(* Logix 5000 project; controller VET 1756-L62 rev 19.52; software revision 19.01; part 7 of 27 *)

        [7].Data.flags[2] := 5, [7].Data.flags[3] := 5, [7].Data.flags[4] := 5, [7].Data.flags[5] := 5, [7].Data.flags[6] := 5, [7].Data.flags[7] := 5, [7].Data.flags[8] := 5, [7].Data.fecha_i[0] := 20140324, [7].Data.fecha_i[1] := 20140324, [7].Data.fecha_i[2] := 20140324, [7].Data.fecha_i[3] := 20140324, [7].Data.fecha_i[4] := 20140324, [7].Data.fecha_i[5] := 20140324, [7].Data.fecha_i[6] := 20140324, [7].Data.fecha_i[7] := 20140324, [7].Data.fecha_i[8] := 20140324, [7].Data.fecha_f[0] := 20140324, [7].Data.fecha_f[1] := 20140324, [7].Data.fecha_f[2] := 20140324, [7].Data.fecha_f[3] := 20140324, [7].Data.fecha_f[4] := 20140324, [7].Data.fecha_f[5] := 20140324, [7].Data.fecha_f[6] := 20140324, [7].Data.fecha_f[7] := 20140324, [7].Data.fecha_f[8] := 20140324, [7].Data.hora_i[0] := 11072683, [7].Data.hora_i[1] := 11073663, [7].Data.hora_i[2] := 11072683, [7].Data.hora_i[3] := 11073503, [7].Data.hora_i[4] := 11072683, [7].Data.hora_i[5] := 11074453, [7].Data.hora_i[6] := 11100033, [7].Data.hora_i[7] := 11072683, [7].Data.hora_i[8] := 11073593, [7].Data.hora_f[0] := 11073623, [7].Data.hora_f[1] := 11074913, [7].Data.hora_f[2] := 11073463, [7].Data.hora_f[3] := 11074613, [7].Data.hora_f[4] := 11074413, [7].Data.hora_f[5] := 11075843, [7].Data.hora_f[6] := 11105503, [7].Data.hora_f[7] := 11073553, [7].Data.hora_f[8] := 11074863, [8].Head.folio := 20, [8].Head.orden := -2, [8].Head.formula := 'DUMMY$00$00$00$00$00', [8].Head.estado := 5, [8].Head.correlativo := 10, [8].Head.total_batch := 10, [8].Head.peso_teorico := 1201.0, [8].Data.codigo[0] := 5, [8].Data.codigo[1] := 6, [8].Data.codigo[2] := 7, [8].Data.codigo[3] := 8, [8].Data.codigo[4] := 10, [8].Data.codigo[5] := 20, [8].Data.codigo[6] := 25, [8].Data.codigo[7] := 49, [8].Data.codigo[8] := 50, [8].Data.peso_f[0] := 8.0,
        [8].Data.peso_f[1] := 7.0, [8].Data.peso_f[2] := 6.0, [8].Data.peso_f[3] := 5.0, [8].Data.peso_f[4] := 600.0, [8].Data.peso_f[5] := 400.0, [8].Data.peso_f[6] := 95.0, [8].Data.peso_f[7] := 30.0, [8].Data.peso_f[8] := 50.0, [9].Head.folio := 21, [9].Head.orden := -3, [9].Head.formula := 'DUMMY$00$00$00$00$00', [9].Head.correlativo := 1, [9].Head.total_batch := 20, [9].Head.peso_teorico := 1733.0, [9].Data.codigo[0] := 51, [9].Data.codigo[1] := 53, [9].Data.codigo[2] := 55, [9].Data.codigo[3] := 57, [9].Data.codigo[4] := 60, [9].Data.codigo[5] := 62, [9].Data.codigo[6] := 64, [9].Data.codigo[7] := 66, [9].Data.codigo[8] := 67, [9].Data.codigo[9] := 68, [9].Data.codigo[10] := 69, [9].Data.codigo[11] := 70, [9].Data.codigo[12] := 74, [9].Data.codigo[13] := 75, [9].Data.codigo[14] := 76, [9].Data.codigo[15] := 77, [9].Data.codigo[16] := 81, [9].Data.peso_f[0] := 400.0, [9].Data.peso_f[1] := 350.0, [9].Data.peso_f[2] := 175.0, [9].Data.peso_f[3] := 225.0, [9].Data.peso_f[4] := 125.0, [9].Data.peso_f[5] := 125.0, [9].Data.peso_f[6] := 65.0, [9].Data.peso_f[7] := 65.0, [9].Data.peso_f[8] := 30.0, [9].Data.peso_f[9] := 25.0, [9].Data.peso_f[10] := 17.5, [9].Data.peso_f[11] := 17.5, [9].Data.peso_f[12] := 30.0, [9].Data.peso_f[13] := 5.0, [9].Data.peso_f[14] := 4.0, [9].Data.peso_f[15] := 4.0, [9].Data.peso_f[16] := 70.0, [9].Data.peso_r[0] := 406.2177, [9].Data.peso_r[1] := 352.48218, [9].Data.peso_r[2] := 181.6532, [9].Data.peso_r[3] := 226.84772, [9].Data.peso_r[4] := 129.14812, [9].Data.peso_r[5] := 129.12715, [9].Data.peso_r[6] := 68.647064, [9].Data.peso_r[7] := 68.64438, [9].Data.peso_r[8] := 30.003521, [9].Data.peso_r[9] := 24.965416, [9].Data.peso_r[10] := 17.580997, [9].Data.peso_r[11] := 17.461937,
        [9].Data.peso_r[12] := 30.00344, [9].Data.peso_r[13] := 4.9946327, [9].Data.peso_r[14] := 3.9117737, [9].Data.peso_r[15] := 3.952877, [9].Data.peso_r[16] := 70.002106, [9].Data.tolva[0] := 2, [9].Data.tolva[1] := 4, [9].Data.tolva[2] := 10, [9].Data.tolva[3] := 12, [9].Data.tolva[4] := 7, [9].Data.tolva[5] := 9, [9].Data.tolva[6] := 15, [9].Data.tolva[7] := 17, [9].Data.tolva[8] := 18, [9].Data.tolva[9] := 19, [9].Data.tolva[10] := 20, [9].Data.tolva[11] := 21, [9].Data.tolva[12] := 26, [9].Data.tolva[13] := 27, [9].Data.tolva[14] := 28, [9].Data.tolva[15] := 29, [9].Data.tolva[16] := 38, [9].Data.lugar[0] := 1, [9].Data.lugar[1] := 1, [9].Data.lugar[2] := 1, [9].Data.lugar[3] := 1, [9].Data.lugar[4] := 2, [9].Data.lugar[5] := 2, [9].Data.lugar[6] := 2, [9].Data.lugar[7] := 2, [9].Data.lugar[8] := 3, [9].Data.lugar[9] := 3, [9].Data.lugar[10] := 3, [9].Data.lugar[11] := 3, [9].Data.lugar[12] := 4, [9].Data.lugar[13] := 4, [9].Data.lugar[14] := 4, [9].Data.lugar[15] := 4, [9].Data.lugar[16] := 6, [9].Data.flags[0] := 5, [9].Data.flags[1] := 5, [9].Data.flags[2] := 5, [9].Data.flags[3] := 5, [9].Data.flags[4] := 5, [9].Data.flags[5] := 5, [9].Data.flags[6] := 5, [9].Data.flags[7] := 5, [9].Data.flags[8] := 5, [9].Data.flags[9] := 5, [9].Data.flags[10] := 5, [9].Data.flags[11] := 5, [9].Data.flags[12] := 5, [9].Data.flags[13] := 5, [9].Data.flags[14] := 5, [9].Data.flags[15] := 5, [9].Data.flags[16] := 5, [9].Data.fecha_i[0] := 20140324, [9].Data.fecha_i[1] := 20140324, [9].Data.fecha_i[2] := 20140324, [9].Data.fecha_i[3] := 20140324,
        [9].Data.fecha_i[4] := 20140324, [9].Data.fecha_i[5] := 20140324, [9].Data.fecha_i[6] := 20140324, [9].Data.fecha_i[7] := 20140324, [9].Data.fecha_i[8] := 20140324, [9].Data.fecha_i[9] := 20140324, [9].Data.fecha_i[10] := 20140324, [9].Data.fecha_i[11] := 20140324, [9].Data.fecha_i[12] := 20140324, [9].Data.fecha_i[13] := 20140324, [9].Data.fecha_i[14] := 20140324, [9].Data.fecha_i[15] := 20140324, [9].Data.fecha_i[16] := 20140324, [9].Data.fecha_f[0] := 20140324, [9].Data.fecha_f[1] := 20140324, [9].Data.fecha_f[2] := 20140324, [9].Data.fecha_f[3] := 20140324, [9].Data.fecha_f[4] := 20140324, [9].Data.fecha_f[5] := 20140324, [9].Data.fecha_f[6] := 20140324, [9].Data.fecha_f[7] := 20140324, [9].Data.fecha_f[8] := 20140324, [9].Data.fecha_f[9] := 20140324, [9].Data.fecha_f[10] := 20140324, [9].Data.fecha_f[11] := 20140324, [9].Data.fecha_f[12] := 20140324, [9].Data.fecha_f[13] := 20140324, [9].Data.fecha_f[14] := 20140324, [9].Data.fecha_f[15] := 20140324, [9].Data.fecha_f[16] := 20140324, [9].Data.hora_i[0] := 15282353, [9].Data.hora_i[1] := 15284663, [9].Data.hora_i[2] := 15290343, [9].Data.hora_i[3] := 15292253, [9].Data.hora_i[4] := 15282353, [9].Data.hora_i[5] := 15284903, [9].Data.hora_i[6] := 15290823, [9].Data.hora_i[7] := 15292083, [9].Data.hora_i[8] := 15282353, [9].Data.hora_i[9] := 15311783, [9].Data.hora_i[10] := 15321493, [9].Data.hora_i[11] := 15325653, [9].Data.hora_i[12] := 15282353, [9].Data.hora_i[13] := 15323253, [9].Data.hora_i[14] := 15324993, [9].Data.hora_i[15] := 15330103, [9].Data.hora_i[16] := 15335763, [9].Data.hora_f[0] := 15284623, [9].Data.hora_f[1] := 15290303, [9].Data.hora_f[2] := 15292213, [9].Data.hora_f[3] := 15294183, [9].Data.hora_f[4] := 15284863, [9].Data.hora_f[5] := 15290783, [9].Data.hora_f[6] := 15292043, [9].Data.hora_f[7] := 15293023, [9].Data.hora_f[8] := 15311743, [9].Data.hora_f[9] := 15321453, [9].Data.hora_f[10] := 15325613, [9].Data.hora_f[11] := 15333843, [9].Data.hora_f[12] := 15323213,
        [9].Data.hora_f[13] := 15324953, [9].Data.hora_f[14] := 15330063, [9].Data.hora_f[15] := 15331563, [9].Data.hora_f[16] := 15344023, [10].Head.folio := 22, [10].Head.orden := -3, [10].Head.formula := 'DUMMY$00$00$00$00$00', [10].Head.correlativo := 2, [10].Head.total_batch := 20, [10].Head.peso_teorico := 1733.0, [10].Data.codigo[0] := 51, [10].Data.codigo[1] := 53, [10].Data.codigo[2] := 55, [10].Data.codigo[3] := 57, [10].Data.codigo[4] := 60, [10].Data.codigo[5] := 62, [10].Data.codigo[6] := 64, [10].Data.codigo[7] := 66, [10].Data.codigo[8] := 67, [10].Data.codigo[9] := 68, [10].Data.codigo[10] := 69, [10].Data.codigo[11] := 70, [10].Data.codigo[12] := 74, [10].Data.codigo[13] := 75, [10].Data.codigo[14] := 76, [10].Data.codigo[15] := 77, [10].Data.codigo[16] := 81, [10].Data.peso_f[0] := 400.0, [10].Data.peso_f[1] := 350.0, [10].Data.peso_f[2] := 175.0, [10].Data.peso_f[3] := 225.0, [10].Data.peso_f[4] := 125.0, [10].Data.peso_f[5] := 125.0, [10].Data.peso_f[6] := 65.0, [10].Data.peso_f[7] := 65.0, [10].Data.peso_f[8] := 30.0, [10].Data.peso_f[9] := 25.0, [10].Data.peso_f[10] := 17.5, [10].Data.peso_f[11] := 17.5, [10].Data.peso_f[12] := 30.0, [10].Data.peso_f[13] := 5.0, [10].Data.peso_f[14] := 4.0, [10].Data.peso_f[15] := 4.0, [10].Data.peso_f[16] := 70.0, [10].Data.peso_r[0] := 406.18576, [10].Data.peso_r[1] := 355.42447, [10].Data.peso_r[2] := 181.19794, [10].Data.peso_r[3] := 226.84515, [10].Data.peso_r[4] := 125.444466, [10].Data.peso_r[5] := 127.34431, [10].Data.peso_r[6] := 68.58177, [10].Data.peso_r[7] := 68.6817, [10].Data.peso_r[8] := 30.003046, [10].Data.peso_r[9] := 24.965014, [10].Data.peso_r[10] := 17.42197, [10].Data.peso_r[11] := 17.461983, [10].Data.peso_r[12] := 30.003046, [10].Data.peso_r[13] := 4.995043, [10].Data.peso_r[14] := 3.9528885, [10].Data.peso_r[15] := 3.9532852,
        [10].Data.peso_r[16] := 70.0021, [10].Data.tolva[0] := 2, [10].Data.tolva[1] := 4, [10].Data.tolva[2] := 10, [10].Data.tolva[3] := 12, [10].Data.tolva[4] := 7, [10].Data.tolva[5] := 9, [10].Data.tolva[6] := 15, [10].Data.tolva[7] := 17, [10].Data.tolva[8] := 18, [10].Data.tolva[9] := 19, [10].Data.tolva[10] := 20, [10].Data.tolva[11] := 21, [10].Data.tolva[12] := 26, [10].Data.tolva[13] := 27, [10].Data.tolva[14] := 28, [10].Data.tolva[15] := 29, [10].Data.tolva[16] := 38, [10].Data.lugar[0] := 1, [10].Data.lugar[1] := 1, [10].Data.lugar[2] := 1, [10].Data.lugar[3] := 1, [10].Data.lugar[4] := 2, [10].Data.lugar[5] := 2, [10].Data.lugar[6] := 2, [10].Data.lugar[7] := 2, [10].Data.lugar[8] := 3, [10].Data.lugar[9] := 3, [10].Data.lugar[10] := 3, [10].Data.lugar[11] := 3, [10].Data.lugar[12] := 4, [10].Data.lugar[13] := 4, [10].Data.lugar[14] := 4, [10].Data.lugar[15] := 4, [10].Data.lugar[16] := 6, [10].Data.flags[0] := 5, [10].Data.flags[1] := 5, [10].Data.flags[2] := 5, [10].Data.flags[3] := 5, [10].Data.flags[4] := 5, [10].Data.flags[5] := 5, [10].Data.flags[6] := 5, [10].Data.flags[7] := 5, [10].Data.flags[8] := 5, [10].Data.flags[9] := 5, [10].Data.flags[10] := 5, [10].Data.flags[11] := 5, [10].Data.flags[12] := 5, [10].Data.flags[13] := 5, [10].Data.flags[14] := 5, [10].Data.flags[15] := 5, [10].Data.flags[16] := 5, [10].Data.fecha_i[0] := 20140324, [10].Data.fecha_i[1] := 20140324, [10].Data.fecha_i[2] := 20140324, [10].Data.fecha_i[3] := 20140324, [10].Data.fecha_i[4] := 20140324, [10].Data.fecha_i[5] := 20140324, [10].Data.fecha_i[6] := 20140324, [10].Data.fecha_i[7] := 20140324,
        [10].Data.fecha_i[8] := 20140324, [10].Data.fecha_i[9] := 20140324, [10].Data.fecha_i[10] := 20140324, [10].Data.fecha_i[11] := 20140324, [10].Data.fecha_i[12] := 20140324, [10].Data.fecha_i[13] := 20140324, [10].Data.fecha_i[14] := 20140324, [10].Data.fecha_i[15] := 20140324, [10].Data.fecha_i[16] := 20140324, [10].Data.fecha_f[0] := 20140324, [10].Data.fecha_f[1] := 20140324, [10].Data.fecha_f[2] := 20140324, [10].Data.fecha_f[3] := 20140324, [10].Data.fecha_f[4] := 20140324, [10].Data.fecha_f[5] := 20140324, [10].Data.fecha_f[6] := 20140324, [10].Data.fecha_f[7] := 20140324, [10].Data.fecha_f[8] := 20140324, [10].Data.fecha_f[9] := 20140324, [10].Data.fecha_f[10] := 20140324, [10].Data.fecha_f[11] := 20140324, [10].Data.fecha_f[12] := 20140324, [10].Data.fecha_f[13] := 20140324, [10].Data.fecha_f[14] := 20140324, [10].Data.fecha_f[15] := 20140324, [10].Data.fecha_f[16] := 20140324, [10].Data.hora_i[0] := 15335773, [10].Data.hora_i[1] := 15342253, [10].Data.hora_i[2] := 15402193, [10].Data.hora_i[3] := 15403953, [10].Data.hora_i[4] := 15335773, [10].Data.hora_i[5] := 15340653, [10].Data.hora_i[6] := 15341983, [10].Data.hora_i[7] := 15343023, [10].Data.hora_i[8] := 15335773, [10].Data.hora_i[9] := 15402173, [10].Data.hora_i[10] := 15411913, [10].Data.hora_i[11] := 15415733, [10].Data.hora_i[12] := 15335773, [10].Data.hora_i[13] := 15350103, [10].Data.hora_i[14] := 15402183, [10].Data.hora_i[15] := 15403313, [10].Data.hora_i[16] := 15425823, [10].Data.hora_f[0] := 15342213, [10].Data.hora_f[1] := 15350583, [10].Data.hora_f[2] := 15403913, [10].Data.hora_f[3] := 15405703, [10].Data.hora_f[4] := 15340613, [10].Data.hora_f[5] := 15341943, [10].Data.hora_f[6] := 15342983, [10].Data.hora_f[7] := 15343963, [10].Data.hora_f[8] := 15350063, [10].Data.hora_f[9] := 15411873, [10].Data.hora_f[10] := 15415693, [10].Data.hora_f[11] := 15423913, [10].Data.hora_f[12] := 15350063, [10].Data.hora_f[13] := 15351773, [10].Data.hora_f[14] := 15403273, [10].Data.hora_f[15] := 15404783, [10].Data.hora_f[16] := 15434053,
        [11].Head.folio := 23, [11].Head.orden := -3, [11].Head.formula := 'DUMMY$00$00$00$00$00', [11].Head.correlativo := 3, [11].Head.total_batch := 20, [11].Head.peso_teorico := 1733.0, [11].Data.codigo[0] := 51, [11].Data.codigo[1] := 53, [11].Data.codigo[2] := 55, [11].Data.codigo[3] := 57, [11].Data.codigo[4] := 60, [11].Data.codigo[5] := 62, [11].Data.codigo[6] := 64, [11].Data.codigo[7] := 66, [11].Data.codigo[8] := 67, [11].Data.codigo[9] := 68, [11].Data.codigo[10] := 69, [11].Data.codigo[11] := 70, [11].Data.codigo[12] := 74, [11].Data.codigo[13] := 75, [11].Data.codigo[14] := 76, [11].Data.codigo[15] := 77, [11].Data.codigo[16] := 81, [11].Data.peso_f[0] := 400.0, [11].Data.peso_f[1] := 350.0, [11].Data.peso_f[2] := 175.0, [11].Data.peso_f[3] := 225.0, [11].Data.peso_f[4] := 125.0, [11].Data.peso_f[5] := 125.0, [11].Data.peso_f[6] := 65.0, [11].Data.peso_f[7] := 65.0, [11].Data.peso_f[8] := 30.0, [11].Data.peso_f[9] := 25.0, [11].Data.peso_f[10] := 17.5, [11].Data.peso_f[11] := 17.5, [11].Data.peso_f[12] := 30.0, [11].Data.peso_f[13] := 5.0, [11].Data.peso_f[14] := 4.0, [11].Data.peso_f[15] := 4.0, [11].Data.peso_f[16] := 70.0, [11].Data.peso_r[0] := 400.25983, [11].Data.peso_r[1] := 352.48248, [11].Data.peso_r[2] := 175.69269, [11].Data.peso_r[3] := 226.84637, [11].Data.peso_r[4] := 125.44443, [11].Data.peso_r[5] := 127.34447, [11].Data.peso_r[6] := 66.7538, [11].Data.peso_r[7] := 64.86154, [11].Data.peso_r[8] := 30.003036, [11].Data.peso_r[9] := 25.005493, [11].Data.peso_r[10] := 17.461853, [11].Data.peso_r[11] := 17.462425, [11].Data.peso_r[12] := 30.003036, [11].Data.peso_r[13] := 4.995037, [11].Data.peso_r[14] := 3.9113045, [11].Data.peso_r[15] := 3.9532928, [11].Data.peso_r[16] := 70.0001, [11].Data.tolva[0] := 2, [11].Data.tolva[1] := 4, [11].Data.tolva[2] := 10,
        [11].Data.tolva[3] := 12, [11].Data.tolva[4] := 7, [11].Data.tolva[5] := 9, [11].Data.tolva[6] := 15, [11].Data.tolva[7] := 17, [11].Data.tolva[8] := 18, [11].Data.tolva[9] := 19, [11].Data.tolva[10] := 20, [11].Data.tolva[11] := 21, [11].Data.tolva[12] := 26, [11].Data.tolva[13] := 27, [11].Data.tolva[14] := 28, [11].Data.tolva[15] := 29, [11].Data.tolva[16] := 38, [11].Data.lugar[0] := 1, [11].Data.lugar[1] := 1, [11].Data.lugar[2] := 1, [11].Data.lugar[3] := 1, [11].Data.lugar[4] := 2, [11].Data.lugar[5] := 2, [11].Data.lugar[6] := 2, [11].Data.lugar[7] := 2, [11].Data.lugar[8] := 3, [11].Data.lugar[9] := 3, [11].Data.lugar[10] := 3, [11].Data.lugar[11] := 3, [11].Data.lugar[12] := 4, [11].Data.lugar[13] := 4, [11].Data.lugar[14] := 4, [11].Data.lugar[15] := 4, [11].Data.lugar[16] := 6, [11].Data.flags[0] := 5, [11].Data.flags[1] := 5, [11].Data.flags[2] := 5, [11].Data.flags[3] := 5, [11].Data.flags[4] := 5, [11].Data.flags[5] := 5, [11].Data.flags[6] := 5, [11].Data.flags[7] := 5, [11].Data.flags[8] := 5, [11].Data.flags[9] := 5, [11].Data.flags[10] := 5, [11].Data.flags[11] := 5, [11].Data.flags[12] := 5, [11].Data.flags[13] := 5, [11].Data.flags[14] := 5, [11].Data.flags[15] := 5, [11].Data.flags[16] := 5, [11].Data.fecha_i[0] := 20140324, [11].Data.fecha_i[1] := 20140324, [11].Data.fecha_i[2] := 20140324, [11].Data.fecha_i[3] := 20140324, [11].Data.fecha_i[4] := 20140324, [11].Data.fecha_i[5] := 20140324, [11].Data.fecha_i[6] := 20140324, [11].Data.fecha_i[7] := 20140324, [11].Data.fecha_i[8] := 20140324, [11].Data.fecha_i[9] := 20140324, [11].Data.fecha_i[10] := 20140324, [11].Data.fecha_i[11] := 20140324,
        [11].Data.fecha_i[12] := 20140324, [11].Data.fecha_i[13] := 20140324, [11].Data.fecha_i[14] := 20140324, [11].Data.fecha_i[15] := 20140324, [11].Data.fecha_i[16] := 20140324, [11].Data.fecha_f[0] := 20140324, [11].Data.fecha_f[1] := 20140324, [11].Data.fecha_f[2] := 20140324, [11].Data.fecha_f[3] := 20140324, [11].Data.fecha_f[4] := 20140324, [11].Data.fecha_f[5] := 20140324, [11].Data.fecha_f[6] := 20140324, [11].Data.fecha_f[7] := 20140324, [11].Data.fecha_f[8] := 20140324, [11].Data.fecha_f[9] := 20140324, [11].Data.fecha_f[10] := 20140324, [11].Data.fecha_f[11] := 20140324, [11].Data.fecha_f[12] := 20140324, [11].Data.fecha_f[13] := 20140324, [11].Data.fecha_f[14] := 20140324, [11].Data.fecha_f[15] := 20140324, [11].Data.fecha_f[16] := 20140324, [11].Data.hora_i[0] := 15425833, [11].Data.hora_i[1] := 15431183, [11].Data.hora_i[2] := 15454413, [11].Data.hora_i[3] := 15455193, [11].Data.hora_i[4] := 15425833, [11].Data.hora_i[5] := 15430713, [11].Data.hora_i[6] := 15454423, [11].Data.hora_i[7] := 15455843, [11].Data.hora_i[8] := 15425833, [11].Data.hora_i[9] := 15440173, [11].Data.hora_i[10] := 15445913, [11].Data.hora_i[11] := 15453733, [11].Data.hora_i[12] := 15425833, [11].Data.hora_i[13] := 15440163, [11].Data.hora_i[14] := 15441903, [11].Data.hora_i[15] := 15443023, [11].Data.hora_i[16] := 15481743, [11].Data.hora_f[0] := 15431143, [11].Data.hora_f[1] := 15454373, [11].Data.hora_f[2] := 15455153, [11].Data.hora_f[3] := 15472663, [11].Data.hora_f[4] := 15430673, [11].Data.hora_f[5] := 15454383, [11].Data.hora_f[6] := 15455803, [11].Data.hora_f[7] := 15460433, [11].Data.hora_f[8] := 15440123, [11].Data.hora_f[9] := 15445873, [11].Data.hora_f[10] := 15453693, [11].Data.hora_f[11] := 15461933, [11].Data.hora_f[12] := 15440123, [11].Data.hora_f[13] := 15441863, [11].Data.hora_f[14] := 15442983, [11].Data.hora_f[15] := 15444513, [11].Data.hora_f[16] := 15485973, [12].Head.folio := 24, [12].Head.orden := -3, [12].Head.formula := 'DUMMY$00$00$00$00$00', [12].Head.correlativo := 4,
        [12].Head.total_batch := 20, [12].Head.peso_teorico := 1733.0, [12].Data.codigo[0] := 51, [12].Data.codigo[1] := 53, [12].Data.codigo[2] := 55, [12].Data.codigo[3] := 57, [12].Data.codigo[4] := 60, [12].Data.codigo[5] := 62, [12].Data.codigo[6] := 64, [12].Data.codigo[7] := 66, [12].Data.codigo[8] := 67, [12].Data.codigo[9] := 68, [12].Data.codigo[10] := 69, [12].Data.codigo[11] := 70, [12].Data.codigo[12] := 74, [12].Data.codigo[13] := 75, [12].Data.codigo[14] := 76, [12].Data.codigo[15] := 77, [12].Data.codigo[16] := 81, [12].Data.peso_f[0] := 400.0, [12].Data.peso_f[1] := 350.0, [12].Data.peso_f[2] := 175.0, [12].Data.peso_f[3] := 225.0, [12].Data.peso_f[4] := 125.0, [12].Data.peso_f[5] := 125.0, [12].Data.peso_f[6] := 65.0, [12].Data.peso_f[7] := 65.0, [12].Data.peso_f[8] := 30.0, [12].Data.peso_f[9] := 25.0, [12].Data.peso_f[10] := 17.5, [12].Data.peso_f[11] := 17.5, [12].Data.peso_f[12] := 30.0, [12].Data.peso_f[13] := 5.0, [12].Data.peso_f[14] := 4.0, [12].Data.peso_f[15] := 4.0, [12].Data.peso_f[16] := 70.0, [12].Data.peso_r[0] := 400.2613, [12].Data.peso_r[1] := 352.48242, [12].Data.peso_r[2] := 175.88062, [12].Data.peso_r[3] := 229.9057, [12].Data.peso_r[4] := 125.44438, [12].Data.peso_r[5] := 127.34422, [12].Data.peso_r[6] := 64.84152, [12].Data.peso_r[7] := 64.861115, [12].Data.peso_r[8] := 30.003, [12].Data.peso_r[9] := 25.005491, [12].Data.peso_r[10] := 17.461853, [12].Data.peso_r[11] := 17.461967, [12].Data.peso_r[12] := 30.003, [12].Data.peso_r[13] := 4.9950314, [12].Data.peso_r[14] := 3.9931755, [12].Data.peso_r[15] := 3.9945488, [12].Data.peso_r[16] := 70.000114, [12].Data.tolva[0] := 2, [12].Data.tolva[1] := 4, [12].Data.tolva[2] := 10, [12].Data.tolva[3] := 12, [12].Data.tolva[4] := 7, [12].Data.tolva[5] := 9, [12].Data.tolva[6] := 15,
        [12].Data.tolva[7] := 17, [12].Data.tolva[8] := 18, [12].Data.tolva[9] := 19, [12].Data.tolva[10] := 20, [12].Data.tolva[11] := 21, [12].Data.tolva[12] := 26, [12].Data.tolva[13] := 27, [12].Data.tolva[14] := 28, [12].Data.tolva[15] := 29, [12].Data.tolva[16] := 38, [12].Data.lugar[0] := 1, [12].Data.lugar[1] := 1, [12].Data.lugar[2] := 1, [12].Data.lugar[3] := 1, [12].Data.lugar[4] := 2, [12].Data.lugar[5] := 2, [12].Data.lugar[6] := 2, [12].Data.lugar[7] := 2, [12].Data.lugar[8] := 3, [12].Data.lugar[9] := 3, [12].Data.lugar[10] := 3, [12].Data.lugar[11] := 3, [12].Data.lugar[12] := 4, [12].Data.lugar[13] := 4, [12].Data.lugar[14] := 4, [12].Data.lugar[15] := 4, [12].Data.lugar[16] := 6, [12].Data.flags[0] := 5, [12].Data.flags[1] := 5, [12].Data.flags[2] := 5, [12].Data.flags[3] := 5, [12].Data.flags[4] := 5, [12].Data.flags[5] := 5, [12].Data.flags[6] := 5, [12].Data.flags[7] := 5, [12].Data.flags[8] := 5, [12].Data.flags[9] := 5, [12].Data.flags[10] := 5, [12].Data.flags[11] := 5, [12].Data.flags[12] := 5, [12].Data.flags[13] := 5, [12].Data.flags[14] := 5, [12].Data.flags[15] := 5, [12].Data.flags[16] := 5, [12].Data.fecha_i[0] := 20140324, [12].Data.fecha_i[1] := 20140324, [12].Data.fecha_i[2] := 20140324, [12].Data.fecha_i[3] := 20140324, [12].Data.fecha_i[4] := 20140324, [12].Data.fecha_i[5] := 20140324, [12].Data.fecha_i[6] := 20140324, [12].Data.fecha_i[7] := 20140324, [12].Data.fecha_i[8] := 20140324, [12].Data.fecha_i[9] := 20140324, [12].Data.fecha_i[10] := 20140324, [12].Data.fecha_i[11] := 20140324, [12].Data.fecha_i[12] := 20140324, [12].Data.fecha_i[13] := 20140324, [12].Data.fecha_i[14] := 20140324, [12].Data.fecha_i[15] := 20140324,
        [12].Data.fecha_i[16] := 20140324, [12].Data.fecha_f[0] := 20140324, [12].Data.fecha_f[1] := 20140324, [12].Data.fecha_f[2] := 20140324, [12].Data.fecha_f[3] := 20140324, [12].Data.fecha_f[4] := 20140324, [12].Data.fecha_f[5] := 20140324, [12].Data.fecha_f[6] := 20140324, [12].Data.fecha_f[7] := 20140324, [12].Data.fecha_f[8] := 20140324, [12].Data.fecha_f[9] := 20140324, [12].Data.fecha_f[10] := 20140324, [12].Data.fecha_f[11] := 20140324, [12].Data.fecha_f[12] := 20140324, [12].Data.fecha_f[13] := 20140324, [12].Data.fecha_f[14] := 20140324, [12].Data.fecha_f[15] := 20140324, [12].Data.fecha_f[16] := 20140324, [12].Data.hora_i[0] := 15481753, [12].Data.hora_i[1] := 15483103, [12].Data.hora_i[2] := 15484333, [12].Data.hora_i[3] := 15485113, [12].Data.hora_i[4] := 15481753, [12].Data.hora_i[5] := 15482633, [12].Data.hora_i[6] := 15510173, [12].Data.hora_i[7] := 15510803, [12].Data.hora_i[8] := 15481753, [12].Data.hora_i[9] := 15492093, [12].Data.hora_i[10] := 15501833, [12].Data.hora_i[11] := 15505663, [12].Data.hora_i[12] := 15481753, [12].Data.hora_i[13] := 15492083, [12].Data.hora_i[14] := 15493823, [12].Data.hora_i[15] := 15494953, [12].Data.hora_i[16] := 15515733, [12].Data.hora_f[0] := 15483063, [12].Data.hora_f[1] := 15484293, [12].Data.hora_f[2] := 15485073, [12].Data.hora_f[3] := 15485993, [12].Data.hora_f[4] := 15482593, [12].Data.hora_f[5] := 15510133, [12].Data.hora_f[6] := 15510763, [12].Data.hora_f[7] := 15511393, [12].Data.hora_f[8] := 15492043, [12].Data.hora_f[9] := 15501793, [12].Data.hora_f[10] := 15505623, [12].Data.hora_f[11] := 15513853, [12].Data.hora_f[12] := 15492043, [12].Data.hora_f[13] := 15493783, [12].Data.hora_f[14] := 15494913, [12].Data.hora_f[15] := 15500473, [12].Data.hora_f[16] := 15523963, [13].Head.folio := 25, [13].Head.orden := -3, [13].Head.formula := 'DUMMY$00$00$00$00$00', [13].Head.correlativo := 5, [13].Head.total_batch := 20, [13].Head.peso_teorico := 1733.0, [13].Data.codigo[0] := 51, [13].Data.codigo[1] := 53,
        [13].Data.codigo[2] := 55, [13].Data.codigo[3] := 57, [13].Data.codigo[4] := 60, [13].Data.codigo[5] := 62, [13].Data.codigo[6] := 64, [13].Data.codigo[7] := 66, [13].Data.codigo[8] := 67, [13].Data.codigo[9] := 68, [13].Data.codigo[10] := 69, [13].Data.codigo[11] := 70, [13].Data.codigo[12] := 74, [13].Data.codigo[13] := 75, [13].Data.codigo[14] := 76, [13].Data.codigo[15] := 77, [13].Data.codigo[16] := 81, [13].Data.peso_f[0] := 400.0, [13].Data.peso_f[1] := 350.0, [13].Data.peso_f[2] := 175.0, [13].Data.peso_f[3] := 225.0, [13].Data.peso_f[4] := 125.0, [13].Data.peso_f[5] := 125.0, [13].Data.peso_f[6] := 65.0, [13].Data.peso_f[7] := 65.0, [13].Data.peso_f[8] := 30.0, [13].Data.peso_f[9] := 25.0, [13].Data.peso_f[10] := 17.5, [13].Data.peso_f[11] := 17.5, [13].Data.peso_f[12] := 30.0, [13].Data.peso_f[13] := 5.0, [13].Data.peso_f[14] := 4.0, [13].Data.peso_f[15] := 4.0, [13].Data.peso_f[16] := 70.0, [13].Data.peso_r[0] := 400.2615, [13].Data.peso_r[1] := 352.48227, [13].Data.peso_r[2] := 175.8805, [13].Data.peso_r[3] := 226.84717, [13].Data.peso_r[4] := 125.44438, [13].Data.peso_r[5] := 127.34419, [13].Data.peso_r[6] := 66.67056, [13].Data.peso_r[7] := 64.86157, [13].Data.peso_r[8] := 30.003036, [13].Data.peso_r[9] := 24.987019, [13].Data.peso_r[10] := 17.463833, [13].Data.peso_r[11] := 17.492538, [13].Data.peso_r[12] := 30.003036, [13].Data.peso_r[13] := 4.9950447, [13].Data.peso_r[14] := 3.9935875, [13].Data.peso_r[15] := 3.9949074, [13].Data.peso_r[16] := 69.50179, [13].Data.tolva[0] := 2, [13].Data.tolva[1] := 4, [13].Data.tolva[2] := 10, [13].Data.tolva[3] := 12, [13].Data.tolva[4] := 7, [13].Data.tolva[5] := 9, [13].Data.tolva[6] := 15, [13].Data.tolva[7] := 17, [13].Data.tolva[8] := 18, [13].Data.tolva[9] := 19, [13].Data.tolva[10] := 20,
        [13].Data.tolva[11] := 21, [13].Data.tolva[12] := 26, [13].Data.tolva[13] := 27, [13].Data.tolva[14] := 28, [13].Data.tolva[15] := 29, [13].Data.tolva[16] := 38, [13].Data.lugar[0] := 1, [13].Data.lugar[1] := 1, [13].Data.lugar[2] := 1, [13].Data.lugar[3] := 1, [13].Data.lugar[4] := 2, [13].Data.lugar[5] := 2, [13].Data.lugar[6] := 2, [13].Data.lugar[7] := 2, [13].Data.lugar[8] := 3, [13].Data.lugar[9] := 3, [13].Data.lugar[10] := 3, [13].Data.lugar[11] := 3, [13].Data.lugar[12] := 4, [13].Data.lugar[13] := 4, [13].Data.lugar[14] := 4, [13].Data.lugar[15] := 4, [13].Data.lugar[16] := 6, [13].Data.flags[0] := 5, [13].Data.flags[1] := 5, [13].Data.flags[2] := 5, [13].Data.flags[3] := 5, [13].Data.flags[4] := 5, [13].Data.flags[5] := 5, [13].Data.flags[6] := 5, [13].Data.flags[7] := 5, [13].Data.flags[8] := 5, [13].Data.flags[9] := 5, [13].Data.flags[10] := 5, [13].Data.flags[11] := 5, [13].Data.flags[12] := 5, [13].Data.flags[13] := 5, [13].Data.flags[14] := 5, [13].Data.flags[15] := 5, [13].Data.flags[16] := 5, [13].Data.fecha_i[0] := 20140324, [13].Data.fecha_i[1] := 20140324, [13].Data.fecha_i[2] := 20140324, [13].Data.fecha_i[3] := 20140324, [13].Data.fecha_i[4] := 20140324, [13].Data.fecha_i[5] := 20140324, [13].Data.fecha_i[6] := 20140324, [13].Data.fecha_i[7] := 20140324, [13].Data.fecha_i[8] := 20140324, [13].Data.fecha_i[9] := 20140324, [13].Data.fecha_i[10] := 20140324, [13].Data.fecha_i[11] := 20140324, [13].Data.fecha_i[12] := 20140324, [13].Data.fecha_i[13] := 20140324, [13].Data.fecha_i[14] := 20140324, [13].Data.fecha_i[15] := 20140324, [13].Data.fecha_i[16] := 20140324, [13].Data.fecha_f[0] := 20140324, [13].Data.fecha_f[1] := 20140324, [13].Data.fecha_f[2] := 20140324,
        [13].Data.fecha_f[3] := 20140324, [13].Data.fecha_f[4] := 20140324, [13].Data.fecha_f[5] := 20140324, [13].Data.fecha_f[6] := 20140324, [13].Data.fecha_f[7] := 20140324, [13].Data.fecha_f[8] := 20140324, [13].Data.fecha_f[9] := 20140324, [13].Data.fecha_f[10] := 20140324, [13].Data.fecha_f[11] := 20140324, [13].Data.fecha_f[12] := 20140324, [13].Data.fecha_f[13] := 20140324, [13].Data.fecha_f[14] := 20140324, [13].Data.fecha_f[15] := 20140324, [13].Data.fecha_f[16] := 20140324, [13].Data.hora_i[0] := 15515743, [13].Data.hora_i[1] := 15521093, [13].Data.hora_i[2] := 15522323, [13].Data.hora_i[3] := 15523113, [13].Data.hora_i[4] := 15515743, [13].Data.hora_i[5] := 15520623, [13].Data.hora_i[6] := 15523103, [13].Data.hora_i[7] := 15524343, [13].Data.hora_i[8] := 15515743, [13].Data.hora_i[9] := 15530083, [13].Data.hora_i[10] := 15535769, [13].Data.hora_i[11] := 15543579, [13].Data.hora_i[12] := 15515743, [13].Data.hora_i[13] := 15530073, [13].Data.hora_i[14] := 15531783, [13].Data.hora_i[15] := 15532913, [13].Data.hora_i[16] := 15553579, [13].Data.hora_f[0] := 15521053, [13].Data.hora_f[1] := 15522283, [13].Data.hora_f[2] := 15523063, [13].Data.hora_f[3] := 15523993, [13].Data.hora_f[4] := 15520583, [13].Data.hora_f[5] := 15523063, [13].Data.hora_f[6] := 15524303, [13].Data.hora_f[7] := 15524933, [13].Data.hora_f[8] := 15530033, [13].Data.hora_f[9] := 15535749, [13].Data.hora_f[10] := 15543559, [13].Data.hora_f[11] := 15551764, [13].Data.hora_f[12] := 15530033, [13].Data.hora_f[13] := 15531743, [13].Data.hora_f[14] := 15532873, [13].Data.hora_f[15] := 15534433, [13].Data.hora_f[16] := 15561754, [14].Head.folio := 26, [14].Head.orden := -3, [14].Head.formula := 'DUMMY$00$00$00$00$00', [14].Head.correlativo := 6, [14].Head.total_batch := 20, [14].Head.peso_teorico := 1733.0, [14].Data.codigo[0] := 51, [14].Data.codigo[1] := 53, [14].Data.codigo[2] := 55, [14].Data.codigo[3] := 57, [14].Data.codigo[4] := 60, [14].Data.codigo[5] := 62,
        [14].Data.codigo[6] := 64, [14].Data.codigo[7] := 66, [14].Data.codigo[8] := 67, [14].Data.codigo[9] := 68, [14].Data.codigo[10] := 69, [14].Data.codigo[11] := 70, [14].Data.codigo[12] := 74, [14].Data.codigo[13] := 75, [14].Data.codigo[14] := 76, [14].Data.codigo[15] := 77, [14].Data.codigo[16] := 81, [14].Data.peso_f[0] := 400.0, [14].Data.peso_f[1] := 350.0, [14].Data.peso_f[2] := 175.0, [14].Data.peso_f[3] := 225.0, [14].Data.peso_f[4] := 125.0, [14].Data.peso_f[5] := 125.0, [14].Data.peso_f[6] := 65.0, [14].Data.peso_f[7] := 65.0, [14].Data.peso_f[8] := 30.0, [14].Data.peso_f[9] := 25.0, [14].Data.peso_f[10] := 17.5, [14].Data.peso_f[11] := 17.5, [14].Data.peso_f[12] := 30.0, [14].Data.peso_f[13] := 5.0, [14].Data.peso_f[14] := 4.0, [14].Data.peso_f[15] := 4.0, [14].Data.peso_f[16] := 70.0, [14].Data.peso_r[0] := 405.18765, [14].Data.peso_r[1] := 347.0085, [14].Data.peso_r[2] := 172.9342, [14].Data.peso_r[3] := 221.31152, [14].Data.peso_r[4] := 125.07125, [14].Data.peso_r[5] := 127.7055, [14].Data.peso_r[6] := 67.87331, [14].Data.peso_r[7] := 65.28912, [14].Data.peso_r[8] := 29.954077, [14].Data.peso_r[9] := 24.973166, [14].Data.peso_r[10] := 17.489925, [14].Data.peso_r[11] := 17.490517, [14].Data.peso_r[12] := 29.954084, [14].Data.peso_r[13] := 4.965147, [14].Data.peso_r[14] := 3.9367218, [14].Data.peso_r[15] := 3.9845467, [14].Data.peso_r[16] := 69.8018, [14].Data.tolva[0] := 2, [14].Data.tolva[1] := 4, [14].Data.tolva[2] := 10, [14].Data.tolva[3] := 12, [14].Data.tolva[4] := 7, [14].Data.tolva[5] := 9, [14].Data.tolva[6] := 15, [14].Data.tolva[7] := 17, [14].Data.tolva[8] := 18, [14].Data.tolva[9] := 19, [14].Data.tolva[10] := 20, [14].Data.tolva[11] := 21, [14].Data.tolva[12] := 26, [14].Data.tolva[13] := 27, [14].Data.tolva[14] := 28,
        [14].Data.tolva[15] := 29, [14].Data.tolva[16] := 38, [14].Data.lugar[0] := 1, [14].Data.lugar[1] := 1, [14].Data.lugar[2] := 1, [14].Data.lugar[3] := 1, [14].Data.lugar[4] := 2, [14].Data.lugar[5] := 2, [14].Data.lugar[6] := 2, [14].Data.lugar[7] := 2, [14].Data.lugar[8] := 3, [14].Data.lugar[9] := 3, [14].Data.lugar[10] := 3, [14].Data.lugar[11] := 3, [14].Data.lugar[12] := 4, [14].Data.lugar[13] := 4, [14].Data.lugar[14] := 4, [14].Data.lugar[15] := 4, [14].Data.lugar[16] := 6, [14].Data.flags[0] := 5, [14].Data.flags[1] := 5, [14].Data.flags[2] := 5, [14].Data.flags[3] := 5, [14].Data.flags[4] := 5, [14].Data.flags[5] := 5, [14].Data.flags[6] := 5, [14].Data.flags[7] := 5, [14].Data.flags[8] := 5, [14].Data.flags[9] := 5, [14].Data.flags[10] := 5, [14].Data.flags[11] := 5, [14].Data.flags[12] := 5, [14].Data.flags[13] := 5, [14].Data.flags[14] := 5, [14].Data.flags[15] := 5, [14].Data.flags[16] := 5, [14].Data.fecha_i[0] := 20140324, [14].Data.fecha_i[1] := 20140324, [14].Data.fecha_i[2] := 20140324, [14].Data.fecha_i[3] := 20140324, [14].Data.fecha_i[4] := 20140324, [14].Data.fecha_i[5] := 20140324, [14].Data.fecha_i[6] := 20140324, [14].Data.fecha_i[7] := 20140324, [14].Data.fecha_i[8] := 20140324, [14].Data.fecha_i[9] := 20140324, [14].Data.fecha_i[10] := 20140324, [14].Data.fecha_i[11] := 20140324, [14].Data.fecha_i[12] := 20140324, [14].Data.fecha_i[13] := 20140324, [14].Data.fecha_i[14] := 20140324, [14].Data.fecha_i[15] := 20140324, [14].Data.fecha_i[16] := 20140324, [14].Data.fecha_f[0] := 20140324, [14].Data.fecha_f[1] := 20140324, [14].Data.fecha_f[2] := 20140324, [14].Data.fecha_f[3] := 20140324, [14].Data.fecha_f[4] := 20140324, [14].Data.fecha_f[5] := 20140324, [14].Data.fecha_f[6] := 20140324,
        [14].Data.fecha_f[7] := 20140324, [14].Data.fecha_f[8] := 20140324, [14].Data.fecha_f[9] := 20140324, [14].Data.fecha_f[10] := 20140324, [14].Data.fecha_f[11] := 20140324, [14].Data.fecha_f[12] := 20140324, [14].Data.fecha_f[13] := 20140324, [14].Data.fecha_f[14] := 20140324, [14].Data.fecha_f[15] := 20140324, [14].Data.fecha_f[16] := 20140324, [14].Data.hora_i[0] := 15553584, [14].Data.hora_i[1] := 15560269, [14].Data.hora_i[2] := 15561464, [14].Data.hora_i[3] := 15562219, [14].Data.hora_i[4] := 15553584, [14].Data.hora_i[5] := 15554444, [14].Data.hora_i[6] := 15561879, [14].Data.hora_i[7] := 15563379, [14].Data.hora_i[8] := 15553584, [14].Data.hora_i[9] := 15563899, [14].Data.hora_i[10] := 15573609, [14].Data.hora_i[11] := 15581424, [14].Data.hora_i[12] := 15553584, [14].Data.hora_i[13] := 15563894, [14].Data.hora_i[14] := 15565604, [14].Data.hora_i[15] := 15570709, [14].Data.hora_i[16] := 15591434, [14].Data.hora_f[0] := 15560249, [14].Data.hora_f[1] := 15561444, [14].Data.hora_f[2] := 15562199, [14].Data.hora_f[3] := 15563089, [14].Data.hora_f[4] := 15554424, [14].Data.hora_f[5] := 15561859, [14].Data.hora_f[6] := 15563359, [14].Data.hora_f[7] := 15563959, [14].Data.hora_f[8] := 15563879, [14].Data.hora_f[9] := 15573589, [14].Data.hora_f[10] := 15581404, [14].Data.hora_f[11] := 15585604, [14].Data.hora_f[12] := 15563874, [14].Data.hora_f[13] := 15565584, [14].Data.hora_f[14] := 15570689, [14].Data.hora_f[15] := 15572179, [14].Data.hora_f[16] := 15595649, [15].Head.folio := 27, [15].Head.orden := -3, [15].Head.formula := 'DUMMY$00$00$00$00$00', [15].Head.correlativo := 7, [15].Head.total_batch := 20, [15].Head.peso_teorico := 1733.0, [15].Data.codigo[0] := 51, [15].Data.codigo[1] := 53, [15].Data.codigo[2] := 55, [15].Data.codigo[3] := 57, [15].Data.codigo[4] := 60, [15].Data.codigo[5] := 62, [15].Data.codigo[6] := 64, [15].Data.codigo[7] := 66, [15].Data.codigo[8] := 67, [15].Data.codigo[9] := 68,
        [15].Data.codigo[10] := 69, [15].Data.codigo[11] := 70, [15].Data.codigo[12] := 74, [15].Data.codigo[13] := 75, [15].Data.codigo[14] := 76, [15].Data.codigo[15] := 77, [15].Data.codigo[16] := 81, [15].Data.peso_f[0] := 400.0, [15].Data.peso_f[1] := 350.0, [15].Data.peso_f[2] := 175.0, [15].Data.peso_f[3] := 225.0, [15].Data.peso_f[4] := 125.0, [15].Data.peso_f[5] := 125.0, [15].Data.peso_f[6] := 65.0, [15].Data.peso_f[7] := 65.0, [15].Data.peso_f[8] := 30.0, [15].Data.peso_f[9] := 25.0, [15].Data.peso_f[10] := 17.5, [15].Data.peso_f[11] := 17.5, [15].Data.peso_f[12] := 30.0, [15].Data.peso_f[13] := 5.0, [15].Data.peso_f[14] := 4.0, [15].Data.peso_f[15] := 4.0, [15].Data.peso_f[16] := 70.0, [15].Data.peso_r[0] := 397.91046, [15].Data.peso_r[1] := 348.57037, [15].Data.peso_r[2] := 173.35175, [15].Data.peso_r[3] := 224.36798, [15].Data.peso_r[4] := 125.071434, [15].Data.peso_r[5] := 128.56516, [15].Data.peso_r[6] := 65.05693, [15].Data.peso_r[7] := 65.05704, [15].Data.peso_r[8] := 29.974127, [15].Data.peso_r[9] := 24.973959, [15].Data.peso_r[10] := 17.489887, [15].Data.peso_r[11] := 17.489935, [15].Data.peso_r[12] := 29.967981, [15].Data.peso_r[13] := 4.9850006, [15].Data.peso_r[14] := 4.004406, [15].Data.peso_r[15] := 4.004547, [15].Data.peso_r[16] := 69.80179, [15].Data.tolva[0] := 2, [15].Data.tolva[1] := 4, [15].Data.tolva[2] := 10, [15].Data.tolva[3] := 12, [15].Data.tolva[4] := 7, [15].Data.tolva[5] := 9, [15].Data.tolva[6] := 15, [15].Data.tolva[7] := 17, [15].Data.tolva[8] := 18, [15].Data.tolva[9] := 19, [15].Data.tolva[10] := 20, [15].Data.tolva[11] := 29, [15].Data.tolva[12] := 26, [15].Data.tolva[13] := 27, [15].Data.tolva[14] := 28, [15].Data.tolva[15] := 21, [15].Data.tolva[16] := 38, [15].Data.lugar[0] := 1, [15].Data.lugar[1] := 1,
        [15].Data.lugar[2] := 1, [15].Data.lugar[3] := 1, [15].Data.lugar[4] := 2, [15].Data.lugar[5] := 2, [15].Data.lugar[6] := 2, [15].Data.lugar[7] := 2, [15].Data.lugar[8] := 3, [15].Data.lugar[9] := 3, [15].Data.lugar[10] := 3, [15].Data.lugar[11] := 4, [15].Data.lugar[12] := 4, [15].Data.lugar[13] := 4, [15].Data.lugar[14] := 4, [15].Data.lugar[15] := 3, [15].Data.lugar[16] := 6, [15].Data.flags[0] := 5, [15].Data.flags[1] := 5, [15].Data.flags[2] := 5, [15].Data.flags[3] := 5, [15].Data.flags[4] := 5, [15].Data.flags[5] := 5, [15].Data.flags[6] := 5, [15].Data.flags[7] := 5, [15].Data.flags[8] := 5, [15].Data.flags[9] := 5, [15].Data.flags[10] := 5, [15].Data.flags[11] := 5, [15].Data.flags[12] := 5, [15].Data.flags[13] := 5, [15].Data.flags[14] := 5, [15].Data.flags[15] := 5, [15].Data.flags[16] := 5, [15].Data.fecha_i[0] := 20140324, [15].Data.fecha_i[1] := 20140324, [15].Data.fecha_i[2] := 20140324, [15].Data.fecha_i[3] := 20140324, [15].Data.fecha_i[4] := 20140324, [15].Data.fecha_i[5] := 20140324, [15].Data.fecha_i[6] := 20140324, [15].Data.fecha_i[7] := 20140324, [15].Data.fecha_i[8] := 20140324, [15].Data.fecha_i[9] := 20140324, [15].Data.fecha_i[10] := 20140324, [15].Data.fecha_i[11] := 20140324, [15].Data.fecha_i[12] := 20140324, [15].Data.fecha_i[13] := 20140324, [15].Data.fecha_i[14] := 20140324, [15].Data.fecha_i[15] := 20140324, [15].Data.fecha_i[16] := 20140324, [15].Data.fecha_f[0] := 20140324, [15].Data.fecha_f[1] := 20140324, [15].Data.fecha_f[2] := 20140324, [15].Data.fecha_f[3] := 20140324, [15].Data.fecha_f[4] := 20140324, [15].Data.fecha_f[5] := 20140324, [15].Data.fecha_f[6] := 20140324, [15].Data.fecha_f[7] := 20140324, [15].Data.fecha_f[8] := 20140324, [15].Data.fecha_f[9] := 20140324, [15].Data.fecha_f[10] := 20140324,
        [15].Data.fecha_f[11] := 20140324, [15].Data.fecha_f[12] := 20140324, [15].Data.fecha_f[13] := 20140324, [15].Data.fecha_f[14] := 20140324, [15].Data.fecha_f[15] := 20140324, [15].Data.fecha_f[16] := 20140324, [15].Data.hora_i[0] := 15592024, [15].Data.hora_i[1] := 15593359, [15].Data.hora_i[2] := 15594569, [15].Data.hora_i[3] := 15595324, [15].Data.hora_i[4] := 15592024, [15].Data.hora_i[5] := 15592884, [15].Data.hora_i[6] := 15595739, [15].Data.hora_i[7] := 16000339, [15].Data.hora_i[8] := 15592024, [15].Data.hora_i[9] := 16002344, [15].Data.hora_i[10] := 16012049, [15].Data.hora_i[11] := 15592024, [15].Data.hora_i[12] := 16000219, [15].Data.hora_i[13] := 16010524, [15].Data.hora_i[14] := 16012204, [15].Data.hora_i[15] := 16015864, [15].Data.hora_i[16] := 16023129, [15].Data.hora_f[0] := 15593339, [15].Data.hora_f[1] := 15594549, [15].Data.hora_f[2] := 15595304, [15].Data.hora_f[3] := 16000199, [15].Data.hora_f[4] := 15592864, [15].Data.hora_f[5] := 15595719, [15].Data.hora_f[6] := 16000319, [15].Data.hora_f[7] := 16000914, [15].Data.hora_f[8] := 16002324, [15].Data.hora_f[9] := 16012029, [15].Data.hora_f[10] := 16015844, [15].Data.hora_f[11] := 16000199, [15].Data.hora_f[12] := 16010504, [15].Data.hora_f[13] := 16012184, [15].Data.hora_f[14] := 16013309, [15].Data.hora_f[15] := 16021349, [15].Data.hora_f[16] := 16031334, [16].Head.folio := 28, [16].Head.orden := -3, [16].Head.formula := 'DUMMY$00$00$00$00$00', [16].Head.correlativo := 8, [16].Head.total_batch := 20, [16].Head.peso_teorico := 1733.0, [16].Data.codigo[0] := 51, [16].Data.codigo[1] := 53, [16].Data.codigo[2] := 55, [16].Data.codigo[3] := 57, [16].Data.codigo[4] := 60, [16].Data.codigo[5] := 62, [16].Data.codigo[6] := 64, [16].Data.codigo[7] := 66, [16].Data.codigo[8] := 67, [16].Data.codigo[9] := 68, [16].Data.codigo[10] := 69, [16].Data.codigo[11] := 70, [16].Data.codigo[12] := 74, [16].Data.codigo[13] := 75,
        [16].Data.codigo[14] := 76, [16].Data.codigo[15] := 77, [16].Data.codigo[16] := 81, [16].Data.peso_f[0] := 400.0, [16].Data.peso_f[1] := 350.0, [16].Data.peso_f[2] := 175.0, [16].Data.peso_f[3] := 225.0, [16].Data.peso_f[4] := 125.0, [16].Data.peso_f[5] := 125.0, [16].Data.peso_f[6] := 65.0, [16].Data.peso_f[7] := 65.0, [16].Data.peso_f[8] := 30.0, [16].Data.peso_f[9] := 25.0, [16].Data.peso_f[10] := 17.5, [16].Data.peso_f[11] := 17.5, [16].Data.peso_f[12] := 30.0, [16].Data.peso_f[13] := 5.0, [16].Data.peso_f[14] := 4.0, [16].Data.peso_f[15] := 4.0, [16].Data.peso_f[16] := 70.0, [16].Data.peso_r[0] := 399.41638, [16].Data.peso_r[1] := 349.9532, [16].Data.peso_r[2] := 173.44592, [16].Data.peso_r[3] := 224.35333, [16].Data.peso_r[4] := 125.06888, [16].Data.peso_r[5] := 127.59076, [16].Data.peso_r[6] := 67.95871, [16].Data.peso_r[7] := 65.37213, [16].Data.peso_r[8] := 29.973724, [16].Data.peso_r[9] := 25.01252, [16].Data.peso_r[10] := 17.487335, [16].Data.peso_r[11] := 17.487408, [16].Data.peso_r[12] := 29.970356, [16].Data.peso_r[13] := 4.9825974, [16].Data.peso_r[14] := 4.00441, [16].Data.peso_r[15] := 4.0045547, [16].Data.peso_r[16] := 70.10178, [16].Data.tolva[0] := 2, [16].Data.tolva[1] := 4, [16].Data.tolva[2] := 10, [16].Data.tolva[3] := 12, [16].Data.tolva[4] := 7, [16].Data.tolva[5] := 9, [16].Data.tolva[6] := 15, [16].Data.tolva[7] := 17, [16].Data.tolva[8] := 18, [16].Data.tolva[9] := 19, [16].Data.tolva[10] := 20, [16].Data.tolva[11] := 29, [16].Data.tolva[12] := 26, [16].Data.tolva[13] := 27, [16].Data.tolva[14] := 28, [16].Data.tolva[15] := 21, [16].Data.tolva[16] := 38, [16].Data.lugar[0] := 1, [16].Data.lugar[1] := 1, [16].Data.lugar[2] := 1, [16].Data.lugar[3] := 1, [16].Data.lugar[4] := 2, [16].Data.lugar[5] := 2,
        [16].Data.lugar[6] := 2, [16].Data.lugar[7] := 2, [16].Data.lugar[8] := 3, [16].Data.lugar[9] := 3, [16].Data.lugar[10] := 3, [16].Data.lugar[11] := 4, [16].Data.lugar[12] := 4, [16].Data.lugar[13] := 4, [16].Data.lugar[14] := 4, [16].Data.lugar[15] := 3, [16].Data.lugar[16] := 6, [16].Data.flags[0] := 5, [16].Data.flags[1] := 5, [16].Data.flags[2] := 5, [16].Data.flags[3] := 5, [16].Data.flags[4] := 5, [16].Data.flags[5] := 5, [16].Data.flags[6] := 5, [16].Data.flags[7] := 5, [16].Data.flags[8] := 5, [16].Data.flags[9] := 5, [16].Data.flags[10] := 5, [16].Data.flags[11] := 5, [16].Data.flags[12] := 5, [16].Data.flags[13] := 5, [16].Data.flags[14] := 5, [16].Data.flags[15] := 5, [16].Data.flags[16] := 5, [16].Data.fecha_i[0] := 20140324, [16].Data.fecha_i[1] := 20140324, [16].Data.fecha_i[2] := 20140324, [16].Data.fecha_i[3] := 20140324, [16].Data.fecha_i[4] := 20140324, [16].Data.fecha_i[5] := 20140324, [16].Data.fecha_i[6] := 20140324, [16].Data.fecha_i[7] := 20140324, [16].Data.fecha_i[8] := 20140324, [16].Data.fecha_i[9] := 20140324, [16].Data.fecha_i[10] := 20140324, [16].Data.fecha_i[11] := 20140324, [16].Data.fecha_i[12] := 20140324, [16].Data.fecha_i[13] := 20140324, [16].Data.fecha_i[14] := 20140324, [16].Data.fecha_i[15] := 20140324, [16].Data.fecha_i[16] := 20140324, [16].Data.fecha_f[0] := 20140324, [16].Data.fecha_f[1] := 20140324, [16].Data.fecha_f[2] := 20140324, [16].Data.fecha_f[3] := 20140324, [16].Data.fecha_f[4] := 20140324, [16].Data.fecha_f[5] := 20140324, [16].Data.fecha_f[6] := 20140324, [16].Data.fecha_f[7] := 20140324, [16].Data.fecha_f[8] := 20140324, [16].Data.fecha_f[9] := 20140324, [16].Data.fecha_f[10] := 20140324, [16].Data.fecha_f[11] := 20140324, [16].Data.fecha_f[12] := 20140324, [16].Data.fecha_f[13] := 20140324, [16].Data.fecha_f[14] := 20140324,
        [16].Data.fecha_f[15] := 20140324, [16].Data.fecha_f[16] := 20140324, [16].Data.hora_i[0] := 16023134, [16].Data.hora_i[1] := 16024474, [16].Data.hora_i[2] := 16025684, [16].Data.hora_i[3] := 16030449, [16].Data.hora_i[4] := 16023134, [16].Data.hora_i[5] := 16023994, [16].Data.hora_i[6] := 16030364, [16].Data.hora_i[7] := 16032219, [16].Data.hora_i[8] := 16023134, [16].Data.hora_i[9] := 16033449, [16].Data.hora_i[10] := 16043169, [16].Data.hora_i[11] := 16023134, [16].Data.hora_i[12] := 16031344, [16].Data.hora_i[13] := 16041654, [16].Data.hora_i[14] := 16043359, [16].Data.hora_i[15] := 16050984, [16].Data.hora_i[16] := 16054269, [16].Data.hora_f[0] := 16024454, [16].Data.hora_f[1] := 16025664, [16].Data.hora_f[2] := 16030429, [16].Data.hora_f[3] := 16031314, [16].Data.hora_f[4] := 16023974, [16].Data.hora_f[5] := 16030344, [16].Data.hora_f[6] := 16032199, [16].Data.hora_f[7] := 16032804, [16].Data.hora_f[8] := 16033429, [16].Data.hora_f[9] := 16043149, [16].Data.hora_f[10] := 16050964, [16].Data.hora_f[11] := 16031324, [16].Data.hora_f[12] := 16041634, [16].Data.hora_f[13] := 16043339, [16].Data.hora_f[14] := 16044464, [16].Data.hora_f[15] := 16052469, [16].Data.hora_f[16] := 16062494, [17].Head.folio := 29, [17].Head.orden := -3, [17].Head.formula := 'DUMMY$00$00$00$00$00', [17].Head.correlativo := 9, [17].Head.total_batch := 20, [17].Head.peso_teorico := 1733.0, [17].Data.codigo[0] := 51, [17].Data.codigo[1] := 53, [17].Data.codigo[2] := 55, [17].Data.codigo[3] := 57, [17].Data.codigo[4] := 60, [17].Data.codigo[5] := 62, [17].Data.codigo[6] := 64, [17].Data.codigo[7] := 66, [17].Data.codigo[8] := 67, [17].Data.codigo[9] := 68, [17].Data.codigo[10] := 69, [17].Data.codigo[11] := 70, [17].Data.codigo[12] := 74, [17].Data.codigo[13] := 75, [17].Data.codigo[14] := 76, [17].Data.codigo[15] := 77, [17].Data.codigo[16] := 81, [17].Data.peso_f[0] := 400.0,
        [17].Data.peso_f[1] := 350.0, [17].Data.peso_f[2] := 175.0, [17].Data.peso_f[3] := 225.0, [17].Data.peso_f[4] := 125.0, [17].Data.peso_f[5] := 125.0, [17].Data.peso_f[6] := 65.0, [17].Data.peso_f[7] := 65.0, [17].Data.peso_f[8] := 30.0, [17].Data.peso_f[9] := 25.0, [17].Data.peso_f[10] := 17.5, [17].Data.peso_f[11] := 17.5, [17].Data.peso_f[12] := 30.0, [17].Data.peso_f[13] := 5.0, [17].Data.peso_f[14] := 4.0, [17].Data.peso_f[15] := 4.0, [17].Data.peso_f[16] := 70.0, [17].Data.peso_r[0] := 399.41718, [17].Data.peso_r[1] := 349.64966, [17].Data.peso_r[2] := 175.0708, [17].Data.peso_r[3] := 225.98505, [17].Data.peso_r[4] := 125.06839, [17].Data.peso_r[5] := 127.61029, [17].Data.peso_r[6] := 65.37216, [17].Data.peso_r[7] := 65.37247, [17].Data.peso_r[8] := 29.994556, [17].Data.peso_r[9] := 25.012424, [17].Data.peso_r[10] := 17.509384, [17].Data.peso_r[11] := 17.509583, [17].Data.peso_r[12] := 29.994267, [17].Data.peso_r[13] := 4.9850388, [17].Data.peso_r[14] := 3.9845657, [17].Data.peso_r[15] := 4.0021057, [17].Data.peso_r[16] := 70.09979, [17].Data.tolva[0] := 2, [17].Data.tolva[1] := 4, [17].Data.tolva[2] := 10, [17].Data.tolva[3] := 12, [17].Data.tolva[4] := 7, [17].Data.tolva[5] := 9, [17].Data.tolva[6] := 15, [17].Data.tolva[7] := 17, [17].Data.tolva[8] := 18, [17].Data.tolva[9] := 19, [17].Data.tolva[10] := 20, [17].Data.tolva[11] := 29, [17].Data.tolva[12] := 26, [17].Data.tolva[13] := 27, [17].Data.tolva[14] := 28, [17].Data.tolva[15] := 21, [17].Data.tolva[16] := 38, [17].Data.lugar[0] := 1, [17].Data.lugar[1] := 1, [17].Data.lugar[2] := 1, [17].Data.lugar[3] := 1, [17].Data.lugar[4] := 2, [17].Data.lugar[5] := 2, [17].Data.lugar[6] := 2, [17].Data.lugar[7] := 2, [17].Data.lugar[8] := 3, [17].Data.lugar[9] := 3,
        [17].Data.lugar[10] := 3, [17].Data.lugar[11] := 4, [17].Data.lugar[12] := 4, [17].Data.lugar[13] := 4, [17].Data.lugar[14] := 4, [17].Data.lugar[15] := 3, [17].Data.lugar[16] := 6, [17].Data.flags[0] := 5, [17].Data.flags[1] := 5, [17].Data.flags[2] := 5, [17].Data.flags[3] := 5, [17].Data.flags[4] := 5, [17].Data.flags[5] := 5, [17].Data.flags[6] := 5, [17].Data.flags[7] := 5, [17].Data.flags[8] := 5, [17].Data.flags[9] := 5, [17].Data.flags[10] := 5, [17].Data.flags[11] := 5, [17].Data.flags[12] := 5, [17].Data.flags[13] := 5, [17].Data.flags[14] := 5, [17].Data.flags[15] := 5, [17].Data.flags[16] := 5, [17].Data.fecha_i[0] := 20140324, [17].Data.fecha_i[1] := 20140324, [17].Data.fecha_i[2] := 20140324, [17].Data.fecha_i[3] := 20140324, [17].Data.fecha_i[4] := 20140324, [17].Data.fecha_i[5] := 20140324, [17].Data.fecha_i[6] := 20140324, [17].Data.fecha_i[7] := 20140324, [17].Data.fecha_i[8] := 20140324, [17].Data.fecha_i[9] := 20140324, [17].Data.fecha_i[10] := 20140324, [17].Data.fecha_i[11] := 20140324, [17].Data.fecha_i[12] := 20140324, [17].Data.fecha_i[13] := 20140324, [17].Data.fecha_i[14] := 20140324, [17].Data.fecha_i[15] := 20140324, [17].Data.fecha_i[16] := 20140324, [17].Data.fecha_f[0] := 20140324, [17].Data.fecha_f[1] := 20140324, [17].Data.fecha_f[2] := 20140324, [17].Data.fecha_f[3] := 20140324, [17].Data.fecha_f[4] := 20140324, [17].Data.fecha_f[5] := 20140324, [17].Data.fecha_f[6] := 20140324, [17].Data.fecha_f[7] := 20140324, [17].Data.fecha_f[8] := 20140324, [17].Data.fecha_f[9] := 20140324, [17].Data.fecha_f[10] := 20140324, [17].Data.fecha_f[11] := 20140324, [17].Data.fecha_f[12] := 20140324, [17].Data.fecha_f[13] := 20140324, [17].Data.fecha_f[14] := 20140324, [17].Data.fecha_f[15] := 20140324, [17].Data.fecha_f[16] := 20140324, [17].Data.hora_i[0] := 16054274, [17].Data.hora_i[1] := 16055619,
        [17].Data.hora_i[2] := 16060824, [17].Data.hora_i[3] := 16061594, [17].Data.hora_i[4] := 16054274, [17].Data.hora_i[5] := 16055134, [17].Data.hora_i[6] := 16061499, [17].Data.hora_i[7] := 16062104, [17].Data.hora_i[8] := 16054274, [17].Data.hora_i[9] := 16064594, [17].Data.hora_i[10] := 16074289, [17].Data.hora_i[11] := 16054274, [17].Data.hora_i[12] := 16062474, [17].Data.hora_i[13] := 16072794, [17].Data.hora_i[14] := 16074489, [17].Data.hora_i[15] := 16082109, [17].Data.hora_i[16] := 16085394, [17].Data.hora_f[0] := 16055599, [17].Data.hora_f[1] := 16060804, [17].Data.hora_f[2] := 16061574, [17].Data.hora_f[3] := 16062469, [17].Data.hora_f[4] := 16055114, [17].Data.hora_f[5] := 16061479, [17].Data.hora_f[6] := 16062084, [17].Data.hora_f[7] := 16062689, [17].Data.hora_f[8] := 16064574, [17].Data.hora_f[9] := 16074269, [17].Data.hora_f[10] := 16082089, [17].Data.hora_f[11] := 16062454, [17].Data.hora_f[12] := 16072774, [17].Data.hora_f[13] := 16074469, [17].Data.hora_f[14] := 16075584, [17].Data.hora_f[15] := 16083599, [17].Data.hora_f[16] := 16093619, [18].Head.folio := 30, [18].Head.orden := -3, [18].Head.formula := 'DUMMY$00$00$00$00$00', [18].Head.correlativo := 10, [18].Head.total_batch := 20, [18].Head.peso_teorico := 1733.0, [18].Data.codigo[0] := 51, [18].Data.codigo[1] := 53, [18].Data.codigo[2] := 55, [18].Data.codigo[3] := 57, [18].Data.codigo[4] := 60, [18].Data.codigo[5] := 62, [18].Data.codigo[6] := 64, [18].Data.codigo[7] := 66, [18].Data.codigo[8] := 67, [18].Data.codigo[9] := 68, [18].Data.codigo[10] := 69, [18].Data.codigo[11] := 70, [18].Data.codigo[12] := 74, [18].Data.codigo[13] := 75, [18].Data.codigo[14] := 76, [18].Data.codigo[15] := 77, [18].Data.codigo[16] := 81, [18].Data.peso_f[0] := 400.0, [18].Data.peso_f[1] := 350.0, [18].Data.peso_f[2] := 175.0, [18].Data.peso_f[3] := 225.0, [18].Data.peso_f[4] := 125.0,
        [18].Data.peso_f[5] := 125.0, [18].Data.peso_f[6] := 65.0, [18].Data.peso_f[7] := 65.0, [18].Data.peso_f[8] := 30.0, [18].Data.peso_f[9] := 25.0, [18].Data.peso_f[10] := 17.5, [18].Data.peso_f[11] := 17.5, [18].Data.peso_f[12] := 30.0, [18].Data.peso_f[13] := 5.0, [18].Data.peso_f[14] := 4.0, [18].Data.peso_f[15] := 4.0, [18].Data.peso_f[16] := 70.0, [18].Data.peso_r[0] := 399.51053, [18].Data.peso_r[1] := 350.04776, [18].Data.peso_r[2] := 175.08862, [18].Data.peso_r[3] := 224.45184, [18].Data.peso_r[4] := 125.070755, [18].Data.peso_r[5] := 125.97429, [18].Data.peso_r[6] := 67.07645, [18].Data.peso_r[7] := 65.28821, [18].Data.peso_r[8] := 29.994556, [18].Data.peso_r[9] := 25.01247, [18].Data.peso_r[10] := 17.506996, [18].Data.peso_r[11] := 17.489944, [18].Data.peso_r[12] := 30.008419, [18].Data.peso_r[13] := 5.005974, [18].Data.peso_r[14] := 4.0019455, [18].Data.peso_r[15] := 4.0045395, [18].Data.peso_r[16] := 69.80178, [18].Data.tolva[0] := 2, [18].Data.tolva[1] := 4, [18].Data.tolva[2] := 10, [18].Data.tolva[3] := 12, [18].Data.tolva[4] := 7, [18].Data.tolva[5] := 9, [18].Data.tolva[6] := 15, [18].Data.tolva[7] := 17, [18].Data.tolva[8] := 18, [18].Data.tolva[9] := 19, [18].Data.tolva[10] := 20, [18].Data.tolva[11] := 29, [18].Data.tolva[12] := 26, [18].Data.tolva[13] := 27, [18].Data.tolva[14] := 28, [18].Data.tolva[15] := 21, [18].Data.tolva[16] := 38, [18].Data.lugar[0] := 1, [18].Data.lugar[1] := 1, [18].Data.lugar[2] := 1, [18].Data.lugar[3] := 1, [18].Data.lugar[4] := 2, [18].Data.lugar[5] := 2, [18].Data.lugar[6] := 2, [18].Data.lugar[7] := 2, [18].Data.lugar[8] := 3, [18].Data.lugar[9] := 3, [18].Data.lugar[10] := 3, [18].Data.lugar[11] := 4, [18].Data.lugar[12] := 4, [18].Data.lugar[13] := 4,
        [18].Data.lugar[14] := 4, [18].Data.lugar[15] := 3, [18].Data.lugar[16] := 6, [18].Data.flags[0] := 5, [18].Data.flags[1] := 5, [18].Data.flags[2] := 5, [18].Data.flags[3] := 5, [18].Data.flags[4] := 5, [18].Data.flags[5] := 5, [18].Data.flags[6] := 5, [18].Data.flags[7] := 5, [18].Data.flags[8] := 5, [18].Data.flags[9] := 5, [18].Data.flags[10] := 5, [18].Data.flags[11] := 5, [18].Data.flags[12] := 5, [18].Data.flags[13] := 5, [18].Data.flags[14] := 5, [18].Data.flags[15] := 5, [18].Data.flags[16] := 5, [18].Data.fecha_i[0] := 20140324, [18].Data.fecha_i[1] := 20140324, [18].Data.fecha_i[2] := 20140324, [18].Data.fecha_i[3] := 20140324, [18].Data.fecha_i[4] := 20140324, [18].Data.fecha_i[5] := 20140324, [18].Data.fecha_i[6] := 20140324, [18].Data.fecha_i[7] := 20140324, [18].Data.fecha_i[8] := 20140324, [18].Data.fecha_i[9] := 20140324, [18].Data.fecha_i[10] := 20140324, [18].Data.fecha_i[11] := 20140324, [18].Data.fecha_i[12] := 20140324, [18].Data.fecha_i[13] := 20140324, [18].Data.fecha_i[14] := 20140324, [18].Data.fecha_i[15] := 20140324, [18].Data.fecha_i[16] := 20140324, [18].Data.fecha_f[0] := 20140324, [18].Data.fecha_f[1] := 20140324, [18].Data.fecha_f[2] := 20140324, [18].Data.fecha_f[3] := 20140324, [18].Data.fecha_f[4] := 20140324, [18].Data.fecha_f[5] := 20140324, [18].Data.fecha_f[6] := 20140324, [18].Data.fecha_f[7] := 20140324, [18].Data.fecha_f[8] := 20140324, [18].Data.fecha_f[9] := 20140324, [18].Data.fecha_f[10] := 20140324, [18].Data.fecha_f[11] := 20140324, [18].Data.fecha_f[12] := 20140324, [18].Data.fecha_f[13] := 20140324, [18].Data.fecha_f[14] := 20140324, [18].Data.fecha_f[15] := 20140324, [18].Data.fecha_f[16] := 20140324, [18].Data.hora_i[0] := 16085399, [18].Data.hora_i[1] := 16090739, [18].Data.hora_i[2] := 16091949, [18].Data.hora_i[3] := 16092709, [18].Data.hora_i[4] := 16085399, [18].Data.hora_i[5] := 16090259,
        [18].Data.hora_i[6] := 16092869, [18].Data.hora_i[7] := 16094579, [18].Data.hora_i[8] := 16085399, [18].Data.hora_i[9] := 16095724, [18].Data.hora_i[10] := 16105449, [18].Data.hora_i[11] := 16085399, [18].Data.hora_i[12] := 16093579, [18].Data.hora_i[13] := 16103894, [18].Data.hora_i[14] := 16105614, [18].Data.hora_i[15] := 16113269, [18].Data.hora_i[16] := 16120549, [18].Data.hora_f[0] := 16090719, [18].Data.hora_f[1] := 16091929, [18].Data.hora_f[2] := 16092689, [18].Data.hora_f[3] := 16093574, [18].Data.hora_f[4] := 16090239, [18].Data.hora_f[5] := 16092849, [18].Data.hora_f[6] := 16094559, [18].Data.hora_f[7] := 16095159, [18].Data.hora_f[8] := 16095704, [18].Data.hora_f[9] := 16105429, [18].Data.hora_f[10] := 16113249, [18].Data.hora_f[11] := 16093559, [18].Data.hora_f[12] := 16103874, [18].Data.hora_f[13] := 16105594, [18].Data.hora_f[14] := 16110714, [18].Data.hora_f[15] := 16114749, [18].Data.hora_f[16] := 16124774, [19].Head.folio := 31, [19].Head.orden := -3, [19].Head.formula := 'DUMMY$00$00$00$00$00', [19].Head.correlativo := 11, [19].Head.total_batch := 20, [19].Head.peso_teorico := 1733.0, [19].Data.codigo[0] := 51, [19].Data.codigo[1] := 53, [19].Data.codigo[2] := 55, [19].Data.codigo[3] := 57, [19].Data.codigo[4] := 60, [19].Data.codigo[5] := 62, [19].Data.codigo[6] := 64, [19].Data.codigo[7] := 66, [19].Data.codigo[8] := 67, [19].Data.codigo[9] := 68, [19].Data.codigo[10] := 69, [19].Data.codigo[11] := 70, [19].Data.codigo[12] := 74, [19].Data.codigo[13] := 75, [19].Data.codigo[14] := 76, [19].Data.codigo[15] := 77, [19].Data.codigo[16] := 81, [19].Data.peso_f[0] := 400.0, [19].Data.peso_f[1] := 350.0, [19].Data.peso_f[2] := 175.0, [19].Data.peso_f[3] := 225.0, [19].Data.peso_f[4] := 125.0, [19].Data.peso_f[5] := 125.0, [19].Data.peso_f[6] := 65.0, [19].Data.peso_f[7] := 65.0, [19].Data.peso_f[8] := 30.0,
        [19].Data.peso_f[9] := 25.0, [19].Data.peso_f[10] := 17.5, [19].Data.peso_f[11] := 17.5, [19].Data.peso_f[12] := 30.0, [19].Data.peso_f[13] := 5.0, [19].Data.peso_f[14] := 4.0, [19].Data.peso_f[15] := 4.0, [19].Data.peso_f[16] := 70.0, [19].Data.peso_r[0] := 398.48602, [19].Data.peso_r[1] := 348.9485, [19].Data.peso_r[2] := 173.54315, [19].Data.peso_r[3] := 223.7793, [19].Data.peso_r[4] := 124.72148, [19].Data.peso_r[5] := 124.674255, [19].Data.peso_r[6] := 67.09276, [19].Data.peso_r[7] := 67.11923, [19].Data.peso_r[8] := 29.992178, [19].Data.peso_r[9] := 25.012426, [19].Data.peso_r[10] := 17.488514, [19].Data.peso_r[11] := 17.50958, [19].Data.peso_r[12] := 29.992468, [19].Data.peso_r[13] := 4.9850464, [19].Data.peso_r[14] := 4.0044594, [19].Data.peso_r[15] := 4.0021286, [19].Data.peso_r[16] := 70.101776, [19].Data.tolva[0] := 2, [19].Data.tolva[1] := 4, [19].Data.tolva[2] := 10, [19].Data.tolva[3] := 12, [19].Data.tolva[4] := 7, [19].Data.tolva[5] := 9, [19].Data.tolva[6] := 15, [19].Data.tolva[7] := 17, [19].Data.tolva[8] := 18, [19].Data.tolva[9] := 19, [19].Data.tolva[10] := 20, [19].Data.tolva[11] := 29, [19].Data.tolva[12] := 26, [19].Data.tolva[13] := 27, [19].Data.tolva[14] := 28, [19].Data.tolva[15] := 21, [19].Data.tolva[16] := 38, [19].Data.lugar[0] := 1, [19].Data.lugar[1] := 1, [19].Data.lugar[2] := 1, [19].Data.lugar[3] := 1, [19].Data.lugar[4] := 2, [19].Data.lugar[5] := 2, [19].Data.lugar[6] := 2, [19].Data.lugar[7] := 2, [19].Data.lugar[8] := 3, [19].Data.lugar[9] := 3, [19].Data.lugar[10] := 3, [19].Data.lugar[11] := 4, [19].Data.lugar[12] := 4, [19].Data.lugar[13] := 4, [19].Data.lugar[14] := 4, [19].Data.lugar[15] := 3, [19].Data.lugar[16] := 6, [19].Data.flags[0] := 5,
        [19].Data.flags[1] := 5, [19].Data.flags[2] := 5, [19].Data.flags[3] := 5, [19].Data.flags[4] := 5, [19].Data.flags[5] := 5, [19].Data.flags[6] := 5, [19].Data.flags[7] := 5, [19].Data.flags[8] := 5, [19].Data.flags[9] := 5, [19].Data.flags[10] := 5, [19].Data.flags[11] := 5, [19].Data.flags[12] := 5, [19].Data.flags[13] := 5, [19].Data.flags[14] := 5, [19].Data.flags[15] := 5, [19].Data.flags[16] := 5, [19].Data.fecha_i[0] := 20140324, [19].Data.fecha_i[1] := 20140324, [19].Data.fecha_i[2] := 20140324, [19].Data.fecha_i[3] := 20140324, [19].Data.fecha_i[4] := 20140324, [19].Data.fecha_i[5] := 20140324, [19].Data.fecha_i[6] := 20140324, [19].Data.fecha_i[7] := 20140324, [19].Data.fecha_i[8] := 20140324, [19].Data.fecha_i[9] := 20140324, [19].Data.fecha_i[10] := 20140324, [19].Data.fecha_i[11] := 20140324, [19].Data.fecha_i[12] := 20140324, [19].Data.fecha_i[13] := 20140324, [19].Data.fecha_i[14] := 20140324, [19].Data.fecha_i[15] := 20140324, [19].Data.fecha_i[16] := 20140324, [19].Data.fecha_f[0] := 20140324, [19].Data.fecha_f[1] := 20140324, [19].Data.fecha_f[2] := 20140324, [19].Data.fecha_f[3] := 20140324, [19].Data.fecha_f[4] := 20140324, [19].Data.fecha_f[5] := 20140324, [19].Data.fecha_f[6] := 20140324, [19].Data.fecha_f[7] := 20140324, [19].Data.fecha_f[8] := 20140324, [19].Data.fecha_f[9] := 20140324, [19].Data.fecha_f[10] := 20140324, [19].Data.fecha_f[11] := 20140324, [19].Data.fecha_f[12] := 20140324, [19].Data.fecha_f[13] := 20140324, [19].Data.fecha_f[14] := 20140324, [19].Data.fecha_f[15] := 20140324, [19].Data.fecha_f[16] := 20140324, [19].Data.hora_i[0] := 16120554, [19].Data.hora_i[1] := 16122259, [19].Data.hora_i[2] := 16123784, [19].Data.hora_i[3] := 16124704, [19].Data.hora_i[4] := 16120554, [19].Data.hora_i[5] := 16121679, [19].Data.hora_i[6] := 16122804, [19].Data.hora_i[7] := 16124769, [19].Data.hora_i[8] := 16120554, [19].Data.hora_i[9] := 16130874,
        [19].Data.hora_i[10] := 16140569, [19].Data.hora_i[11] := 16120554, [19].Data.hora_i[12] := 16124754, [19].Data.hora_i[13] := 16135074, [19].Data.hora_i[14] := 16140769, [19].Data.hora_i[15] := 16144384, [19].Data.hora_i[16] := 16151659, [19].Data.hora_f[0] := 16122239, [19].Data.hora_f[1] := 16123764, [19].Data.hora_f[2] := 16124684, [19].Data.hora_f[3] := 16125774, [19].Data.hora_f[4] := 16121659, [19].Data.hora_f[5] := 16122784, [19].Data.hora_f[6] := 16124749, [19].Data.hora_f[7] := 16130609, [19].Data.hora_f[8] := 16130854, [19].Data.hora_f[9] := 16140549, [19].Data.hora_f[10] := 16144364, [19].Data.hora_f[11] := 16124734, [19].Data.hora_f[12] := 16135054, [19].Data.hora_f[13] := 16140749, [19].Data.hora_f[14] := 16141869, [19].Data.hora_f[15] := 16145879, [19].Data.hora_f[16] := 16155864, [20].Head.folio := 32, [20].Head.orden := -3, [20].Head.formula := 'DUMMY$00$00$00$00$00', [20].Head.correlativo := 12, [20].Head.total_batch := 20, [20].Head.peso_teorico := 1733.0, [20].Data.codigo[0] := 51, [20].Data.codigo[1] := 53, [20].Data.codigo[2] := 55, [20].Data.codigo[3] := 57, [20].Data.codigo[4] := 60, [20].Data.codigo[5] := 62, [20].Data.codigo[6] := 64, [20].Data.codigo[7] := 66, [20].Data.codigo[8] := 67, [20].Data.codigo[9] := 68, [20].Data.codigo[10] := 69, [20].Data.codigo[11] := 70, [20].Data.codigo[12] := 74, [20].Data.codigo[13] := 75, [20].Data.codigo[14] := 76, [20].Data.codigo[15] := 77, [20].Data.codigo[16] := 81, [20].Data.peso_f[0] := 400.0, [20].Data.peso_f[1] := 350.0, [20].Data.peso_f[2] := 175.0, [20].Data.peso_f[3] := 225.0, [20].Data.peso_f[4] := 125.0, [20].Data.peso_f[5] := 125.0, [20].Data.peso_f[6] := 65.0, [20].Data.peso_f[7] := 65.0, [20].Data.peso_f[8] := 30.0, [20].Data.peso_f[9] := 25.0, [20].Data.peso_f[10] := 17.5, [20].Data.peso_f[11] := 17.5, [20].Data.peso_f[12] := 30.0,
        [20].Data.peso_f[13] := 5.0, [20].Data.peso_f[14] := 4.0, [20].Data.peso_f[15] := 4.0, [20].Data.peso_f[16] := 70.0, [20].Data.peso_r[0] := 399.5826, [20].Data.peso_r[1] := 348.13077, [20].Data.peso_r[2] := 174.59515, [20].Data.peso_r[3] := 225.03009, [20].Data.peso_r[4] := 124.72399, [20].Data.peso_r[5] := 124.656075, [20].Data.peso_r[6] := 64.778625, [20].Data.peso_r[7] := 64.712494, [20].Data.peso_r[8] := 30.014198, [20].Data.peso_r[9] := 25.012432, [20].Data.peso_r[10] := 17.509579, [20].Data.peso_r[11] := 17.509575, [20].Data.peso_r[12] := 30.013912, [20].Data.peso_r[13] := 5.0060196, [20].Data.peso_r[14] := 4.0019455, [20].Data.peso_r[15] := 4.004524, [20].Data.peso_r[16] := 70.10178, [20].Data.tolva[0] := 2, [20].Data.tolva[1] := 4, [20].Data.tolva[2] := 10, [20].Data.tolva[3] := 12, [20].Data.tolva[4] := 7, [20].Data.tolva[5] := 9, [20].Data.tolva[6] := 15, [20].Data.tolva[7] := 17, [20].Data.tolva[8] := 18, [20].Data.tolva[9] := 19, [20].Data.tolva[10] := 20, [20].Data.tolva[11] := 29, [20].Data.tolva[12] := 26, [20].Data.tolva[13] := 27, [20].Data.tolva[14] := 28, [20].Data.tolva[15] := 21, [20].Data.tolva[16] := 38, [20].Data.lugar[0] := 1, [20].Data.lugar[1] := 1, [20].Data.lugar[2] := 1, [20].Data.lugar[3] := 1, [20].Data.lugar[4] := 2, [20].Data.lugar[5] := 2, [20].Data.lugar[6] := 2, [20].Data.lugar[7] := 2, [20].Data.lugar[8] := 3, [20].Data.lugar[9] := 3, [20].Data.lugar[10] := 3, [20].Data.lugar[11] := 4, [20].Data.lugar[12] := 4, [20].Data.lugar[13] := 4, [20].Data.lugar[14] := 4, [20].Data.lugar[15] := 3, [20].Data.lugar[16] := 6, [20].Data.flags[0] := 5, [20].Data.flags[1] := 5, [20].Data.flags[2] := 5, [20].Data.flags[3] := 5, [20].Data.flags[4] := 5,
        [20].Data.flags[5] := 5, [20].Data.flags[6] := 5, [20].Data.flags[7] := 5, [20].Data.flags[8] := 5, [20].Data.flags[9] := 5, [20].Data.flags[10] := 5, [20].Data.flags[11] := 5, [20].Data.flags[12] := 5, [20].Data.flags[13] := 5, [20].Data.flags[14] := 5, [20].Data.flags[15] := 5, [20].Data.flags[16] := 5, [20].Data.fecha_i[0] := 20140324, [20].Data.fecha_i[1] := 20140324, [20].Data.fecha_i[2] := 20140324, [20].Data.fecha_i[3] := 20140324, [20].Data.fecha_i[4] := 20140324, [20].Data.fecha_i[5] := 20140324, [20].Data.fecha_i[6] := 20140324, [20].Data.fecha_i[7] := 20140324, [20].Data.fecha_i[8] := 20140324, [20].Data.fecha_i[9] := 20140324, [20].Data.fecha_i[10] := 20140324, [20].Data.fecha_i[11] := 20140324, [20].Data.fecha_i[12] := 20140324, [20].Data.fecha_i[13] := 20140324, [20].Data.fecha_i[14] := 20140324, [20].Data.fecha_i[15] := 20140324, [20].Data.fecha_i[16] := 20140324, [20].Data.fecha_f[0] := 20140324, [20].Data.fecha_f[1] := 20140324, [20].Data.fecha_f[2] := 20140324, [20].Data.fecha_f[3] := 20140324, [20].Data.fecha_f[4] := 20140324, [20].Data.fecha_f[5] := 20140324, [20].Data.fecha_f[6] := 20140324, [20].Data.fecha_f[7] := 20140324, [20].Data.fecha_f[8] := 20140324, [20].Data.fecha_f[9] := 20140324, [20].Data.fecha_f[10] := 20140324, [20].Data.fecha_f[11] := 20140324, [20].Data.fecha_f[12] := 20140324, [20].Data.fecha_f[13] := 20140324, [20].Data.fecha_f[14] := 20140324, [20].Data.fecha_f[15] := 20140324, [20].Data.fecha_f[16] := 20140324, [20].Data.hora_i[0] := 16151664, [20].Data.hora_i[1] := 16153379, [20].Data.hora_i[2] := 16154909, [20].Data.hora_i[3] := 16155834, [20].Data.hora_i[4] := 16151664, [20].Data.hora_i[5] := 16152789, [20].Data.hora_i[6] := 16153904, [20].Data.hora_i[7] := 16154639, [20].Data.hora_i[8] := 16151664, [20].Data.hora_i[9] := 16161989, [20].Data.hora_i[10] := 16171699, [20].Data.hora_i[11] := 16151664, [20].Data.hora_i[12] := 16155864, [20].Data.hora_i[13] := 16170189,
        [20].Data.hora_i[14] := 16171894, [20].Data.hora_i[15] := 16175524, [20].Data.hora_i[16] := 16182814, [20].Data.hora_f[0] := 16153359, [20].Data.hora_f[1] := 16154889, [20].Data.hora_f[2] := 16155814, [20].Data.hora_f[3] := 16160919, [20].Data.hora_f[4] := 16152769, [20].Data.hora_f[5] := 16153884, [20].Data.hora_f[6] := 16154619, [20].Data.hora_f[7] := 16155354, [20].Data.hora_f[8] := 16161969, [20].Data.hora_f[9] := 16171679, [20].Data.hora_f[10] := 16175504, [20].Data.hora_f[11] := 16155844, [20].Data.hora_f[12] := 16170169, [20].Data.hora_f[13] := 16171874, [20].Data.hora_f[14] := 16172994, [20].Data.hora_f[15] := 16181029, [20].Data.hora_f[16] := 16191014, [21].Head.folio := 33, [21].Head.orden := -3, [21].Head.formula := 'DUMMY$00$00$00$00$00', [21].Head.correlativo := 13, [21].Head.total_batch := 20, [21].Head.peso_teorico := 1733.0, [21].Data.codigo[0] := 51, [21].Data.codigo[1] := 53, [21].Data.codigo[2] := 55, [21].Data.codigo[3] := 57, [21].Data.codigo[4] := 60, [21].Data.codigo[5] := 62, [21].Data.codigo[6] := 64, [21].Data.codigo[7] := 66, [21].Data.codigo[8] := 67, [21].Data.codigo[9] := 68, [21].Data.codigo[10] := 69, [21].Data.codigo[11] := 70, [21].Data.codigo[12] := 74, [21].Data.codigo[13] := 75, [21].Data.codigo[14] := 76, [21].Data.codigo[15] := 77, [21].Data.codigo[16] := 81, [21].Data.peso_f[0] := 400.0, [21].Data.peso_f[1] := 350.0, [21].Data.peso_f[2] := 175.0, [21].Data.peso_f[3] := 225.0, [21].Data.peso_f[4] := 125.0, [21].Data.peso_f[5] := 125.0, [21].Data.peso_f[6] := 65.0, [21].Data.peso_f[7] := 65.0, [21].Data.peso_f[8] := 30.0, [21].Data.peso_f[9] := 25.0, [21].Data.peso_f[10] := 17.5, [21].Data.peso_f[11] := 17.5, [21].Data.peso_f[12] := 30.0, [21].Data.peso_f[13] := 5.0, [21].Data.peso_f[14] := 4.0, [21].Data.peso_f[15] := 4.0, [21].Data.peso_f[16] := 70.0,
        [21].Data.peso_r[0] := 399.58627, [21].Data.peso_r[1] := 350.3245, [21].Data.peso_r[2] := 174.66821, [21].Data.peso_r[3] := 224.95996, [21].Data.peso_r[4] := 124.67244, [21].Data.peso_r[5] := 125.35693, [21].Data.peso_r[6] := 67.126724, [21].Data.peso_r[7] := 66.486664, [21].Data.peso_r[8] := 29.99456, [21].Data.peso_r[9] := 24.99279, [21].Data.peso_r[10] := 17.502876, [21].Data.peso_r[11] := 17.470299, [21].Data.peso_r[12] := 29.994236, [21].Data.peso_r[13] := 4.9850273, [21].Data.peso_r[14] := 4.0043945, [21].Data.peso_r[15] := 4.002121, [21].Data.peso_r[16] := 70.101776, [21].Data.tolva[0] := 2, [21].Data.tolva[1] := 4, [21].Data.tolva[2] := 10, [21].Data.tolva[3] := 12, [21].Data.tolva[4] := 7, [21].Data.tolva[5] := 9, [21].Data.tolva[6] := 15, [21].Data.tolva[7] := 17, [21].Data.tolva[8] := 18, [21].Data.tolva[9] := 19, [21].Data.tolva[10] := 20, [21].Data.tolva[11] := 29, [21].Data.tolva[12] := 26, [21].Data.tolva[13] := 27, [21].Data.tolva[14] := 28, [21].Data.tolva[15] := 21, [21].Data.tolva[16] := 38, [21].Data.lugar[0] := 1, [21].Data.lugar[1] := 1, [21].Data.lugar[2] := 1, [21].Data.lugar[3] := 1, [21].Data.lugar[4] := 2, [21].Data.lugar[5] := 2, [21].Data.lugar[6] := 2, [21].Data.lugar[7] := 2, [21].Data.lugar[8] := 3, [21].Data.lugar[9] := 3, [21].Data.lugar[10] := 3, [21].Data.lugar[11] := 4, [21].Data.lugar[12] := 4, [21].Data.lugar[13] := 4, [21].Data.lugar[14] := 4, [21].Data.lugar[15] := 3, [21].Data.lugar[16] := 6, [21].Data.flags[0] := 5, [21].Data.flags[1] := 5, [21].Data.flags[2] := 5, [21].Data.flags[3] := 5, [21].Data.flags[4] := 5, [21].Data.flags[5] := 5, [21].Data.flags[6] := 5, [21].Data.flags[7] := 5, [21].Data.flags[8] := 5,
        [21].Data.flags[9] := 5, [21].Data.flags[10] := 5, [21].Data.flags[11] := 5, [21].Data.flags[12] := 5, [21].Data.flags[13] := 5, [21].Data.flags[14] := 5, [21].Data.flags[15] := 5, [21].Data.flags[16] := 5, [21].Data.fecha_i[0] := 20140324, [21].Data.fecha_i[1] := 20140324, [21].Data.fecha_i[2] := 20140324, [21].Data.fecha_i[3] := 20140324, [21].Data.fecha_i[4] := 20140324, [21].Data.fecha_i[5] := 20140324, [21].Data.fecha_i[6] := 20140324, [21].Data.fecha_i[7] := 20140324, [21].Data.fecha_i[8] := 20140324, [21].Data.fecha_i[9] := 20140324, [21].Data.fecha_i[10] := 20140324, [21].Data.fecha_i[11] := 20140324, [21].Data.fecha_i[12] := 20140324, [21].Data.fecha_i[13] := 20140324, [21].Data.fecha_i[14] := 20140324, [21].Data.fecha_i[15] := 20140324, [21].Data.fecha_i[16] := 20140324, [21].Data.fecha_f[0] := 20140324, [21].Data.fecha_f[1] := 20140324, [21].Data.fecha_f[2] := 20140324, [21].Data.fecha_f[3] := 20140324, [21].Data.fecha_f[4] := 20140324, [21].Data.fecha_f[5] := 20140324, [21].Data.fecha_f[6] := 20140324, [21].Data.fecha_f[7] := 20140324, [21].Data.fecha_f[8] := 20140324, [21].Data.fecha_f[9] := 20140324, [21].Data.fecha_f[10] := 20140324, [21].Data.fecha_f[11] := 20140324, [21].Data.fecha_f[12] := 20140324, [21].Data.fecha_f[13] := 20140324, [21].Data.fecha_f[14] := 20140324, [21].Data.fecha_f[15] := 20140324, [21].Data.fecha_f[16] := 20140324, [21].Data.hora_i[0] := 16182819, [21].Data.hora_i[1] := 16184529, [21].Data.hora_i[2] := 16190059, [21].Data.hora_i[3] := 16190989, [21].Data.hora_i[4] := 16182819, [21].Data.hora_i[5] := 16183944, [21].Data.hora_i[6] := 16185074, [21].Data.hora_i[7] := 16190694, [21].Data.hora_i[8] := 16182819, [21].Data.hora_i[9] := 16193144, [21].Data.hora_i[10] := 16202844, [21].Data.hora_i[11] := 16182819, [21].Data.hora_i[12] := 16191029, [21].Data.hora_i[13] := 16201339, [21].Data.hora_i[14] := 16203049, [21].Data.hora_i[15] := 16210664, [21].Data.hora_i[16] := 16213939, [21].Data.hora_f[0] := 16184509,
        [21].Data.hora_f[1] := 16190039, [21].Data.hora_f[2] := 16190969, [21].Data.hora_f[3] := 16192064, [21].Data.hora_f[4] := 16183924, [21].Data.hora_f[5] := 16185054, [21].Data.hora_f[6] := 16190674, [21].Data.hora_f[7] := 16192524, [21].Data.hora_f[8] := 16193124, [21].Data.hora_f[9] := 16202824, [21].Data.hora_f[10] := 16210644, [21].Data.hora_f[11] := 16191009, [21].Data.hora_f[12] := 16201319, [21].Data.hora_f[13] := 16203029, [21].Data.hora_f[14] := 16204149, [21].Data.hora_f[15] := 16212159, [21].Data.hora_f[16] := 16222134, [22].Head.folio := 34, [22].Head.orden := -3, [22].Head.formula := 'DUMMY$00$00$00$00$00', [22].Head.correlativo := 14, [22].Head.total_batch := 20, [22].Head.peso_teorico := 1733.0, [22].Data.codigo[0] := 51, [22].Data.codigo[1] := 53, [22].Data.codigo[2] := 55, [22].Data.codigo[3] := 57, [22].Data.codigo[4] := 60, [22].Data.codigo[5] := 62, [22].Data.codigo[6] := 64, [22].Data.codigo[7] := 66, [22].Data.codigo[8] := 67, [22].Data.codigo[9] := 68, [22].Data.codigo[10] := 69, [22].Data.codigo[11] := 70, [22].Data.codigo[12] := 74, [22].Data.codigo[13] := 75, [22].Data.codigo[14] := 76, [22].Data.codigo[15] := 77, [22].Data.codigo[16] := 81, [22].Data.peso_f[0] := 400.0, [22].Data.peso_f[1] := 350.0, [22].Data.peso_f[2] := 175.0, [22].Data.peso_f[3] := 225.0, [22].Data.peso_f[4] := 125.0, [22].Data.peso_f[5] := 125.0, [22].Data.peso_f[6] := 65.0, [22].Data.peso_f[7] := 65.0, [22].Data.peso_f[8] := 30.0, [22].Data.peso_f[9] := 25.0, [22].Data.peso_f[10] := 17.5, [22].Data.peso_f[11] := 17.5, [22].Data.peso_f[12] := 30.0, [22].Data.peso_f[13] := 5.0, [22].Data.peso_f[14] := 4.0, [22].Data.peso_f[15] := 4.0, [22].Data.peso_f[16] := 70.0, [22].Data.peso_r[0] := 399.5824, [22].Data.peso_r[1] := 348.13104, [22].Data.peso_r[2] := 174.59534, [22].Data.peso_r[3] := 225.02997,
        [22].Data.peso_r[4] := 124.72398, [22].Data.peso_r[5] := 125.27002, [22].Data.peso_r[6] := 65.37816, [22].Data.peso_r[7] := 65.33685, [22].Data.peso_r[8] := 29.994602, [22].Data.peso_r[9] := 25.01196, [22].Data.peso_r[10] := 17.489922, [22].Data.peso_r[11] := 17.509577, [22].Data.peso_r[12] := 30.013876, [22].Data.peso_r[13] := 5.025734, [22].Data.peso_r[14] := 3.9952278, [22].Data.peso_r[15] := 3.984726, [22].Data.peso_r[16] := 70.10178, [22].Data.tolva[0] := 2, [22].Data.tolva[1] := 4, [22].Data.tolva[2] := 10, [22].Data.tolva[3] := 12, [22].Data.tolva[4] := 7, [22].Data.tolva[5] := 9, [22].Data.tolva[6] := 15, [22].Data.tolva[7] := 17, [22].Data.tolva[8] := 18, [22].Data.tolva[9] := 19, [22].Data.tolva[10] := 20, [22].Data.tolva[11] := 29, [22].Data.tolva[12] := 26, [22].Data.tolva[13] := 27, [22].Data.tolva[14] := 28, [22].Data.tolva[15] := 21, [22].Data.tolva[16] := 38, [22].Data.lugar[0] := 1, [22].Data.lugar[1] := 1, [22].Data.lugar[2] := 1, [22].Data.lugar[3] := 1, [22].Data.lugar[4] := 2, [22].Data.lugar[5] := 2, [22].Data.lugar[6] := 2, [22].Data.lugar[7] := 2, [22].Data.lugar[8] := 3, [22].Data.lugar[9] := 3, [22].Data.lugar[10] := 3, [22].Data.lugar[11] := 4, [22].Data.lugar[12] := 4, [22].Data.lugar[13] := 4, [22].Data.lugar[14] := 4, [22].Data.lugar[15] := 3, [22].Data.lugar[16] := 6, [22].Data.flags[0] := 5, [22].Data.flags[1] := 5, [22].Data.flags[2] := 5, [22].Data.flags[3] := 5, [22].Data.flags[4] := 5, [22].Data.flags[5] := 5, [22].Data.flags[6] := 5, [22].Data.flags[7] := 5, [22].Data.flags[8] := 5, [22].Data.flags[9] := 5, [22].Data.flags[10] := 5, [22].Data.flags[11] := 5, [22].Data.flags[12] := 5,
        [22].Data.flags[13] := 5, [22].Data.flags[14] := 5, [22].Data.flags[15] := 5, [22].Data.flags[16] := 5, [22].Data.fecha_i[0] := 20140324, [22].Data.fecha_i[1] := 20140324, [22].Data.fecha_i[2] := 20140324, [22].Data.fecha_i[3] := 20140324, [22].Data.fecha_i[4] := 20140324, [22].Data.fecha_i[5] := 20140324, [22].Data.fecha_i[6] := 20140324, [22].Data.fecha_i[7] := 20140324, [22].Data.fecha_i[8] := 20140324, [22].Data.fecha_i[9] := 20140324, [22].Data.fecha_i[10] := 20140324, [22].Data.fecha_i[11] := 20140324, [22].Data.fecha_i[12] := 20140324, [22].Data.fecha_i[13] := 20140324, [22].Data.fecha_i[14] := 20140324, [22].Data.fecha_i[15] := 20140324, [22].Data.fecha_i[16] := 20140324, [22].Data.fecha_f[0] := 20140324, [22].Data.fecha_f[1] := 20140324, [22].Data.fecha_f[2] := 20140324, [22].Data.fecha_f[3] := 20140324, [22].Data.fecha_f[4] := 20140324, [22].Data.fecha_f[5] := 20140324, [22].Data.fecha_f[6] := 20140324, [22].Data.fecha_f[7] := 20140324, [22].Data.fecha_f[8] := 20140324, [22].Data.fecha_f[9] := 20140324, [22].Data.fecha_f[10] := 20140324, [22].Data.fecha_f[11] := 20140324, [22].Data.fecha_f[12] := 20140324, [22].Data.fecha_f[13] := 20140324, [22].Data.fecha_f[14] := 20140324, [22].Data.fecha_f[15] := 20140324, [22].Data.fecha_f[16] := 20140324, [22].Data.hora_i[0] := 16213944, [22].Data.hora_i[1] := 16215659, [22].Data.hora_i[2] := 16221189, [22].Data.hora_i[3] := 16222114, [22].Data.hora_i[4] := 16213944, [22].Data.hora_i[5] := 16215069, [22].Data.hora_i[6] := 16220189, [22].Data.hora_i[7] := 16220929, [22].Data.hora_i[8] := 16213944, [22].Data.hora_i[9] := 16224269, [22].Data.hora_i[10] := 16233979, [22].Data.hora_i[11] := 16213944, [22].Data.hora_i[12] := 16222144, [22].Data.hora_i[13] := 16232469, [22].Data.hora_i[14] := 16234179, [22].Data.hora_i[15] := 16241794, [22].Data.hora_i[16] := 16245049, [22].Data.hora_f[0] := 16215639, [22].Data.hora_f[1] := 16221169, [22].Data.hora_f[2] := 16222094, [22].Data.hora_f[3] := 16223199, [22].Data.hora_f[4] := 16215049,
        [22].Data.hora_f[5] := 16220169, [22].Data.hora_f[6] := 16220909, [22].Data.hora_f[7] := 16221644, [22].Data.hora_f[8] := 16224249, [22].Data.hora_f[9] := 16233959, [22].Data.hora_f[10] := 16241774, [22].Data.hora_f[11] := 16222124, [22].Data.hora_f[12] := 16232449, [22].Data.hora_f[13] := 16234159, [22].Data.hora_f[14] := 16235274, [22].Data.hora_f[15] := 16243264, [22].Data.hora_f[16] := 16253259, [23].Head.folio := 35, [23].Head.orden := -3, [23].Head.formula := 'DUMMY$00$00$00$00$00', [23].Head.correlativo := 15, [23].Head.total_batch := 20, [23].Head.peso_teorico := 1733.0, [23].Data.codigo[0] := 51, [23].Data.codigo[1] := 53, [23].Data.codigo[2] := 55, [23].Data.codigo[3] := 57, [23].Data.codigo[4] := 60, [23].Data.codigo[5] := 62, [23].Data.codigo[6] := 64, [23].Data.codigo[7] := 66, [23].Data.codigo[8] := 67, [23].Data.codigo[9] := 68, [23].Data.codigo[10] := 69, [23].Data.codigo[11] := 70, [23].Data.codigo[12] := 74, [23].Data.codigo[13] := 75, [23].Data.codigo[14] := 76, [23].Data.codigo[15] := 77, [23].Data.codigo[16] := 81, [23].Data.peso_f[0] := 400.0, [23].Data.peso_f[1] := 350.0, [23].Data.peso_f[2] := 175.0, [23].Data.peso_f[3] := 225.0, [23].Data.peso_f[4] := 125.0, [23].Data.peso_f[5] := 125.0, [23].Data.peso_f[6] := 65.0, [23].Data.peso_f[7] := 65.0, [23].Data.peso_f[8] := 30.0, [23].Data.peso_f[9] := 25.0, [23].Data.peso_f[10] := 17.5, [23].Data.peso_f[11] := 17.5, [23].Data.peso_f[12] := 30.0, [23].Data.peso_f[13] := 5.0, [23].Data.peso_f[14] := 4.0, [23].Data.peso_f[15] := 4.0, [23].Data.peso_f[16] := 70.0, [23].Data.peso_r[0] := 399.58582, [23].Data.peso_r[1] := 350.33508, [23].Data.peso_r[2] := 173.47327, [23].Data.peso_r[3] := 225.03406, [23].Data.peso_r[4] := 124.72148, [23].Data.peso_r[5] := 124.67212, [23].Data.peso_r[6] := 65.3784, [23].Data.peso_r[7] := 65.37808,
        [23].Data.peso_r[8] := 30.014185, [23].Data.peso_r[9] := 24.992853, [23].Data.peso_r[10] := 17.507015, [23].Data.peso_r[11] := 17.507053, [23].Data.peso_r[12] := 29.99292, [23].Data.peso_r[13] := 5.0035934, [23].Data.peso_r[14] := 4.004406, [23].Data.peso_r[15] := 4.004547, [23].Data.peso_r[16] := 69.80177, [23].Data.tolva[0] := 2, [23].Data.tolva[1] := 4, [23].Data.tolva[2] := 10, [23].Data.tolva[3] := 12, [23].Data.tolva[4] := 7, [23].Data.tolva[5] := 9, [23].Data.tolva[6] := 15, [23].Data.tolva[7] := 17, [23].Data.tolva[8] := 18, [23].Data.tolva[9] := 19, [23].Data.tolva[10] := 20, [23].Data.tolva[11] := 29, [23].Data.tolva[12] := 26, [23].Data.tolva[13] := 27, [23].Data.tolva[14] := 28, [23].Data.tolva[15] := 21, [23].Data.tolva[16] := 38, [23].Data.lugar[0] := 1, [23].Data.lugar[1] := 1, [23].Data.lugar[2] := 1, [23].Data.lugar[3] := 1, [23].Data.lugar[4] := 2, [23].Data.lugar[5] := 2, [23].Data.lugar[6] := 2, [23].Data.lugar[7] := 2, [23].Data.lugar[8] := 3, [23].Data.lugar[9] := 3, [23].Data.lugar[10] := 3, [23].Data.lugar[11] := 4, [23].Data.lugar[12] := 4, [23].Data.lugar[13] := 4, [23].Data.lugar[14] := 4, [23].Data.lugar[15] := 3, [23].Data.lugar[16] := 6, [23].Data.flags[0] := 5, [23].Data.flags[1] := 5, [23].Data.flags[2] := 5, [23].Data.flags[3] := 5, [23].Data.flags[4] := 5, [23].Data.flags[5] := 5, [23].Data.flags[6] := 5, [23].Data.flags[7] := 5, [23].Data.flags[8] := 5, [23].Data.flags[9] := 5, [23].Data.flags[10] := 5, [23].Data.flags[11] := 5, [23].Data.flags[12] := 5, [23].Data.flags[13] := 5, [23].Data.flags[14] := 5, [23].Data.flags[15] := 5, [23].Data.flags[16] := 5,
        [23].Data.fecha_i[0] := 20140324, [23].Data.fecha_i[1] := 20140324, [23].Data.fecha_i[2] := 20140324, [23].Data.fecha_i[3] := 20140324, [23].Data.fecha_i[4] := 20140324, [23].Data.fecha_i[5] := 20140324, [23].Data.fecha_i[6] := 20140324, [23].Data.fecha_i[7] := 20140324, [23].Data.fecha_i[8] := 20140324, [23].Data.fecha_i[9] := 20140324, [23].Data.fecha_i[10] := 20140324, [23].Data.fecha_i[11] := 20140324, [23].Data.fecha_i[12] := 20140324, [23].Data.fecha_i[13] := 20140324, [23].Data.fecha_i[14] := 20140324, [23].Data.fecha_i[15] := 20140324, [23].Data.fecha_i[16] := 20140324, [23].Data.fecha_f[0] := 20140324, [23].Data.fecha_f[1] := 20140324, [23].Data.fecha_f[2] := 20140324, [23].Data.fecha_f[3] := 20140324, [23].Data.fecha_f[4] := 20140324, [23].Data.fecha_f[5] := 20140324, [23].Data.fecha_f[6] := 20140324, [23].Data.fecha_f[7] := 20140324, [23].Data.fecha_f[8] := 20140324, [23].Data.fecha_f[9] := 20140324, [23].Data.fecha_f[10] := 20140324, [23].Data.fecha_f[11] := 20140324, [23].Data.fecha_f[12] := 20140324, [23].Data.fecha_f[13] := 20140324, [23].Data.fecha_f[14] := 20140324, [23].Data.fecha_f[15] := 20140324, [23].Data.fecha_f[16] := 20140324, [23].Data.hora_i[0] := 16245054, [23].Data.hora_i[1] := 16250769, [23].Data.hora_i[2] := 16252309, [23].Data.hora_i[3] := 16253229, [23].Data.hora_i[4] := 16245054, [23].Data.hora_i[5] := 16250179, [23].Data.hora_i[6] := 16251304, [23].Data.hora_i[7] := 16252049, [23].Data.hora_i[8] := 16245054, [23].Data.hora_i[9] := 16255384, [23].Data.hora_i[10] := 16265084, [23].Data.hora_i[11] := 16245054, [23].Data.hora_i[12] := 16253269, [23].Data.hora_i[13] := 16263579, [23].Data.hora_i[14] := 16265284, [23].Data.hora_i[15] := 16272909, [23].Data.hora_i[16] := 16280174, [23].Data.hora_f[0] := 16250749, [23].Data.hora_f[1] := 16252289, [23].Data.hora_f[2] := 16253209, [23].Data.hora_f[3] := 16254309, [23].Data.hora_f[4] := 16250159, [23].Data.hora_f[5] := 16251284, [23].Data.hora_f[6] := 16252029, [23].Data.hora_f[7] := 16252764, [23].Data.hora_f[8] := 16255364,
        [23].Data.hora_f[9] := 16265064, [23].Data.hora_f[10] := 16272889, [23].Data.hora_f[11] := 16253249, [23].Data.hora_f[12] := 16263559, [23].Data.hora_f[13] := 16265264, [23].Data.hora_f[14] := 16270384, [23].Data.hora_f[15] := 16274389, [23].Data.hora_f[16] := 16284369, [24].Head.folio := 36, [24].Head.orden := -3, [24].Head.formula := 'DUMMY$00$00$00$00$00', [24].Head.correlativo := 16, [24].Head.total_batch := 20, [24].Head.peso_teorico := 1733.0, [24].Data.codigo[0] := 51, [24].Data.codigo[1] := 53, [24].Data.codigo[2] := 55, [24].Data.codigo[3] := 57, [24].Data.codigo[4] := 60, [24].Data.codigo[5] := 62, [24].Data.codigo[6] := 64, [24].Data.codigo[7] := 66, [24].Data.codigo[8] := 67, [24].Data.codigo[9] := 68, [24].Data.codigo[10] := 69, [24].Data.codigo[11] := 70, [24].Data.codigo[12] := 74, [24].Data.codigo[13] := 75, [24].Data.codigo[14] := 76, [24].Data.codigo[15] := 77, [24].Data.codigo[16] := 81, [24].Data.peso_f[0] := 400.0, [24].Data.peso_f[1] := 350.0, [24].Data.peso_f[2] := 175.0, [24].Data.peso_f[3] := 225.0, [24].Data.peso_f[4] := 125.0, [24].Data.peso_f[5] := 125.0, [24].Data.peso_f[6] := 65.0, [24].Data.peso_f[7] := 65.0, [24].Data.peso_f[8] := 30.0, [24].Data.peso_f[9] := 25.0, [24].Data.peso_f[10] := 17.5, [24].Data.peso_f[11] := 17.5, [24].Data.peso_f[12] := 30.0, [24].Data.peso_f[13] := 5.0, [24].Data.peso_f[14] := 4.0, [24].Data.peso_f[15] := 4.0, [24].Data.peso_f[16] := 70.0, [24].Data.peso_r[0] := 400.74274, [24].Data.peso_r[1] := 350.04797, [24].Data.peso_r[2] := 175.83899, [24].Data.peso_r[3] := 224.96124, [24].Data.peso_r[4] := 124.67249, [24].Data.peso_r[5] := 125.35711, [24].Data.peso_r[6] := 65.37897, [24].Data.peso_r[7] := 65.18332, [24].Data.peso_r[8] := 29.994566, [24].Data.peso_r[9] := 25.012415, [24].Data.peso_r[10] := 17.509384, [24].Data.peso_r[11] := 17.509583,
        [24].Data.peso_r[12] := 30.013866, [24].Data.peso_r[13] := 4.9850273, [24].Data.peso_r[14] := 4.0043945, [24].Data.peso_r[15] := 4.002121, [24].Data.peso_r[16] := 70.10178, [24].Data.tolva[0] := 2, [24].Data.tolva[1] := 4, [24].Data.tolva[2] := 10, [24].Data.tolva[3] := 12, [24].Data.tolva[4] := 7, [24].Data.tolva[5] := 9, [24].Data.tolva[6] := 15, [24].Data.tolva[7] := 17, [24].Data.tolva[8] := 18, [24].Data.tolva[9] := 19, [24].Data.tolva[10] := 20, [24].Data.tolva[11] := 29, [24].Data.tolva[12] := 26, [24].Data.tolva[13] := 27, [24].Data.tolva[14] := 28, [24].Data.tolva[15] := 21, [24].Data.tolva[16] := 38, [24].Data.lugar[0] := 1, [24].Data.lugar[1] := 1, [24].Data.lugar[2] := 1, [24].Data.lugar[3] := 1, [24].Data.lugar[4] := 2, [24].Data.lugar[5] := 2, [24].Data.lugar[6] := 2, [24].Data.lugar[7] := 2, [24].Data.lugar[8] := 3, [24].Data.lugar[9] := 3, [24].Data.lugar[10] := 3, [24].Data.lugar[11] := 4, [24].Data.lugar[12] := 4, [24].Data.lugar[13] := 4, [24].Data.lugar[14] := 4, [24].Data.lugar[15] := 3, [24].Data.lugar[16] := 6, [24].Data.flags[0] := 5, [24].Data.flags[1] := 5, [24].Data.flags[2] := 5, [24].Data.flags[3] := 5, [24].Data.flags[4] := 5, [24].Data.flags[5] := 5, [24].Data.flags[6] := 5, [24].Data.flags[7] := 5, [24].Data.flags[8] := 5, [24].Data.flags[9] := 5, [24].Data.flags[10] := 5, [24].Data.flags[11] := 5, [24].Data.flags[12] := 5, [24].Data.flags[13] := 5, [24].Data.flags[14] := 5, [24].Data.flags[15] := 5, [24].Data.flags[16] := 5, [24].Data.fecha_i[0] := 20140324, [24].Data.fecha_i[1] := 20140324, [24].Data.fecha_i[2] := 20140324, [24].Data.fecha_i[3] := 20140324,
        [24].Data.fecha_i[4] := 20140324, [24].Data.fecha_i[5] := 20140324, [24].Data.fecha_i[6] := 20140324, [24].Data.fecha_i[7] := 20140324, [24].Data.fecha_i[8] := 20140324, [24].Data.fecha_i[9] := 20140324, [24].Data.fecha_i[10] := 20140324, [24].Data.fecha_i[11] := 20140324, [24].Data.fecha_i[12] := 20140324, [24].Data.fecha_i[13] := 20140324, [24].Data.fecha_i[14] := 20140324, [24].Data.fecha_i[15] := 20140324, [24].Data.fecha_i[16] := 20140324, [24].Data.fecha_f[0] := 20140324, [24].Data.fecha_f[1] := 20140324, [24].Data.fecha_f[2] := 20140324, [24].Data.fecha_f[3] := 20140324, [24].Data.fecha_f[4] := 20140324, [24].Data.fecha_f[5] := 20140324, [24].Data.fecha_f[6] := 20140324, [24].Data.fecha_f[7] := 20140324, [24].Data.fecha_f[8] := 20140324, [24].Data.fecha_f[9] := 20140324, [24].Data.fecha_f[10] := 20140324, [24].Data.fecha_f[11] := 20140324, [24].Data.fecha_f[12] := 20140324, [24].Data.fecha_f[13] := 20140324, [24].Data.fecha_f[14] := 20140324, [24].Data.fecha_f[15] := 20140324, [24].Data.fecha_f[16] := 20140324, [24].Data.hora_i[0] := 16280179, [24].Data.hora_i[1] := 16281899, [24].Data.hora_i[2] := 16283429, [24].Data.hora_i[3] := 16284354, [24].Data.hora_i[4] := 16280179, [24].Data.hora_i[5] := 16281309, [24].Data.hora_i[6] := 16282434, [24].Data.hora_i[7] := 16283174, [24].Data.hora_i[8] := 16280179, [24].Data.hora_i[9] := 16290504, [24].Data.hora_i[10] := 16300209, [24].Data.hora_i[11] := 16280179, [24].Data.hora_i[12] := 16284394, [24].Data.hora_i[13] := 16294719, [24].Data.hora_i[14] := 16300409, [24].Data.hora_i[15] := 16304029, [24].Data.hora_i[16] := 16311299, [24].Data.hora_f[0] := 16281879, [24].Data.hora_f[1] := 16283409, [24].Data.hora_f[2] := 16284334, [24].Data.hora_f[3] := 16285439, [24].Data.hora_f[4] := 16281289, [24].Data.hora_f[5] := 16282414, [24].Data.hora_f[6] := 16283154, [24].Data.hora_f[7] := 16283889, [24].Data.hora_f[8] := 16290484, [24].Data.hora_f[9] := 16300189, [24].Data.hora_f[10] := 16304009, [24].Data.hora_f[11] := 16284374, [24].Data.hora_f[12] := 16294699,
        [24].Data.hora_f[13] := 16300389, [24].Data.hora_f[14] := 16301509, [24].Data.hora_f[15] := 16305519, [24].Data.hora_f[16] := 16315504, [25].Head.folio := 37, [25].Head.orden := -3, [25].Head.formula := 'DUMMY$00$00$00$00$00', [25].Head.correlativo := 17, [25].Head.total_batch := 20, [25].Head.peso_teorico := 1733.0, [25].Data.codigo[0] := 51, [25].Data.codigo[1] := 53, [25].Data.codigo[2] := 55, [25].Data.codigo[3] := 57, [25].Data.codigo[4] := 60, [25].Data.codigo[5] := 62, [25].Data.codigo[6] := 64, [25].Data.codigo[7] := 66, [25].Data.codigo[8] := 67, [25].Data.codigo[9] := 68, [25].Data.codigo[10] := 69, [25].Data.codigo[11] := 70, [25].Data.codigo[12] := 74, [25].Data.codigo[13] := 75, [25].Data.codigo[14] := 76, [25].Data.codigo[15] := 77, [25].Data.codigo[16] := 81, [25].Data.peso_f[0] := 400.0, [25].Data.peso_f[1] := 350.0, [25].Data.peso_f[2] := 175.0, [25].Data.peso_f[3] := 225.0, [25].Data.peso_f[4] := 125.0, [25].Data.peso_f[5] := 125.0, [25].Data.peso_f[6] := 65.0, [25].Data.peso_f[7] := 65.0, [25].Data.peso_f[8] := 30.0, [25].Data.peso_f[9] := 25.0, [25].Data.peso_f[10] := 17.5, [25].Data.peso_f[11] := 17.5, [25].Data.peso_f[12] := 30.0, [25].Data.peso_f[13] := 5.0, [25].Data.peso_f[14] := 4.0, [25].Data.peso_f[15] := 4.0, [25].Data.peso_f[16] := 70.0, [25].Data.peso_r[0] := 400.7444, [25].Data.peso_r[1] := 350.3944, [25].Data.peso_r[2] := 175.42316, [25].Data.peso_r[3] := 225.02997, [25].Data.peso_r[4] := 125.35698, [25].Data.peso_r[5] := 124.72095, [25].Data.peso_r[6] := 65.32411, [25].Data.peso_r[7] := 65.17859, [25].Data.peso_r[8] := 30.014194, [25].Data.peso_r[9] := 24.973179, [25].Data.peso_r[10] := 17.50956, [25].Data.peso_r[11] := 17.509584, [25].Data.peso_r[12] := 29.993803, [25].Data.peso_r[13] := 5.025738, [25].Data.peso_r[14] := 3.9952278, [25].Data.peso_r[15] := 4.0045547,
        [25].Data.peso_r[16] := 70.10178, [25].Data.tolva[0] := 2, [25].Data.tolva[1] := 4, [25].Data.tolva[2] := 10, [25].Data.tolva[3] := 12, [25].Data.tolva[4] := 7, [25].Data.tolva[5] := 9, [25].Data.tolva[6] := 15, [25].Data.tolva[7] := 17, [25].Data.tolva[8] := 18, [25].Data.tolva[9] := 19, [25].Data.tolva[10] := 20, [25].Data.tolva[11] := 29, [25].Data.tolva[12] := 26, [25].Data.tolva[13] := 27, [25].Data.tolva[14] := 28, [25].Data.tolva[15] := 21, [25].Data.tolva[16] := 38, [25].Data.lugar[0] := 1, [25].Data.lugar[1] := 1, [25].Data.lugar[2] := 1, [25].Data.lugar[3] := 1, [25].Data.lugar[4] := 2, [25].Data.lugar[5] := 2, [25].Data.lugar[6] := 2, [25].Data.lugar[7] := 2, [25].Data.lugar[8] := 3, [25].Data.lugar[9] := 3, [25].Data.lugar[10] := 3, [25].Data.lugar[11] := 4, [25].Data.lugar[12] := 4, [25].Data.lugar[13] := 4, [25].Data.lugar[14] := 4, [25].Data.lugar[15] := 3, [25].Data.lugar[16] := 6, [25].Data.flags[0] := 5, [25].Data.flags[1] := 5, [25].Data.flags[2] := 5, [25].Data.flags[3] := 5, [25].Data.flags[4] := 5, [25].Data.flags[5] := 5, [25].Data.flags[6] := 5, [25].Data.flags[7] := 5, [25].Data.flags[8] := 5, [25].Data.flags[9] := 5, [25].Data.flags[10] := 5, [25].Data.flags[11] := 5, [25].Data.flags[12] := 5, [25].Data.flags[13] := 5, [25].Data.flags[14] := 5, [25].Data.flags[15] := 5, [25].Data.flags[16] := 5, [25].Data.fecha_i[0] := 20140324, [25].Data.fecha_i[1] := 20140324, [25].Data.fecha_i[2] := 20140324, [25].Data.fecha_i[3] := 20140324, [25].Data.fecha_i[4] := 20140324, [25].Data.fecha_i[5] := 20140324, [25].Data.fecha_i[6] := 20140324, [25].Data.fecha_i[7] := 20140324,
        [25].Data.fecha_i[8] := 20140324, [25].Data.fecha_i[9] := 20140324, [25].Data.fecha_i[10] := 20140324, [25].Data.fecha_i[11] := 20140324, [25].Data.fecha_i[12] := 20140324, [25].Data.fecha_i[13] := 20140324, [25].Data.fecha_i[14] := 20140324, [25].Data.fecha_i[15] := 20140324, [25].Data.fecha_i[16] := 20140324, [25].Data.fecha_f[0] := 20140324, [25].Data.fecha_f[1] := 20140324, [25].Data.fecha_f[2] := 20140324, [25].Data.fecha_f[3] := 20140324, [25].Data.fecha_f[4] := 20140324, [25].Data.fecha_f[5] := 20140324, [25].Data.fecha_f[6] := 20140324, [25].Data.fecha_f[7] := 20140324, [25].Data.fecha_f[8] := 20140324, [25].Data.fecha_f[9] := 20140324, [25].Data.fecha_f[10] := 20140324, [25].Data.fecha_f[11] := 20140324, [25].Data.fecha_f[12] := 20140324, [25].Data.fecha_f[13] := 20140324, [25].Data.fecha_f[14] := 20140324, [25].Data.fecha_f[15] := 20140324, [25].Data.fecha_f[16] := 20140324, [25].Data.hora_i[0] := 16311304, [25].Data.hora_i[1] := 16313019, [25].Data.hora_i[2] := 16314554, [25].Data.hora_i[3] := 16315479, [25].Data.hora_i[4] := 16311304, [25].Data.hora_i[5] := 16312434, [25].Data.hora_i[6] := 16313554, [25].Data.hora_i[7] := 16314299, [25].Data.hora_i[8] := 16311304, [25].Data.hora_i[9] := 16321629, [25].Data.hora_i[10] := 16331329, [25].Data.hora_i[11] := 16311304, [25].Data.hora_i[12] := 16315504, [25].Data.hora_i[13] := 16325824, [25].Data.hora_i[14] := 16331539, [25].Data.hora_i[15] := 16335149, [25].Data.hora_i[16] := 16342409, [25].Data.hora_f[0] := 16312999, [25].Data.hora_f[1] := 16314534, [25].Data.hora_f[2] := 16315459, [25].Data.hora_f[3] := 16320564, [25].Data.hora_f[4] := 16312414, [25].Data.hora_f[5] := 16313534, [25].Data.hora_f[6] := 16314279, [25].Data.hora_f[7] := 16315014, [25].Data.hora_f[8] := 16321609, [25].Data.hora_f[9] := 16331309, [25].Data.hora_f[10] := 16335129, [25].Data.hora_f[11] := 16315484, [25].Data.hora_f[12] := 16325804, [25].Data.hora_f[13] := 16331519, [25].Data.hora_f[14] := 16332634, [25].Data.hora_f[15] := 16340624, [25].Data.hora_f[16] := 16350629,
        [26].Head.folio := 38, [26].Head.orden := -3, [26].Head.formula := 'DUMMY$00$00$00$00$00', [26].Head.correlativo := 18, [26].Head.total_batch := 20, [26].Head.peso_teorico := 1733.0, [26].Data.codigo[0] := 51, [26].Data.codigo[1] := 53, [26].Data.codigo[2] := 55, [26].Data.codigo[3] := 57, [26].Data.codigo[4] := 60, [26].Data.codigo[5] := 62, [26].Data.codigo[6] := 64, [26].Data.codigo[7] := 66, [26].Data.codigo[8] := 67, [26].Data.codigo[9] := 68, [26].Data.codigo[10] := 69, [26].Data.codigo[11] := 70, [26].Data.codigo[12] := 74, [26].Data.codigo[13] := 75, [26].Data.codigo[14] := 76, [26].Data.codigo[15] := 77, [26].Data.codigo[16] := 81, [26].Data.peso_f[0] := 400.0, [26].Data.peso_f[1] := 350.0, [26].Data.peso_f[2] := 175.0, [26].Data.peso_f[3] := 225.0, [26].Data.peso_f[4] := 125.0, [26].Data.peso_f[5] := 125.0, [26].Data.peso_f[6] := 65.0, [26].Data.peso_f[7] := 65.0, [26].Data.peso_f[8] := 30.0, [26].Data.peso_f[9] := 25.0, [26].Data.peso_f[10] := 17.5, [26].Data.peso_f[11] := 17.5, [26].Data.peso_f[12] := 30.0, [26].Data.peso_f[13] := 5.0, [26].Data.peso_f[14] := 4.0, [26].Data.peso_f[15] := 4.0, [26].Data.peso_f[16] := 70.0, [26].Data.peso_r[0] := 399.58493, [26].Data.peso_r[1] := 350.33487, [26].Data.peso_r[2] := 174.30615, [26].Data.peso_r[3] := 225.03406, [26].Data.peso_r[4] := 125.359535, [26].Data.peso_r[5] := 124.6722, [26].Data.peso_r[6] := 64.77112, [26].Data.peso_r[7] := 64.771484, [26].Data.peso_r[8] := 29.994562, [26].Data.peso_r[9] := 25.012465, [26].Data.peso_r[10] := 17.506996, [26].Data.peso_r[11] := 17.50707, [26].Data.peso_r[12] := 30.01259, [26].Data.peso_r[13] := 5.0035515, [26].Data.peso_r[14] := 4.004402, [26].Data.peso_r[15] := 4.004547, [26].Data.peso_r[16] := 69.801796, [26].Data.tolva[0] := 2, [26].Data.tolva[1] := 4, [26].Data.tolva[2] := 10,
        [26].Data.tolva[3] := 12, [26].Data.tolva[4] := 7, [26].Data.tolva[5] := 9, [26].Data.tolva[6] := 15, [26].Data.tolva[7] := 17, [26].Data.tolva[8] := 18, [26].Data.tolva[9] := 19, [26].Data.tolva[10] := 20, [26].Data.tolva[11] := 29, [26].Data.tolva[12] := 26, [26].Data.tolva[13] := 27, [26].Data.tolva[14] := 28, [26].Data.tolva[15] := 21, [26].Data.tolva[16] := 38, [26].Data.lugar[0] := 1, [26].Data.lugar[1] := 1, [26].Data.lugar[2] := 1, [26].Data.lugar[3] := 1, [26].Data.lugar[4] := 2, [26].Data.lugar[5] := 2, [26].Data.lugar[6] := 2, [26].Data.lugar[7] := 2, [26].Data.lugar[8] := 3, [26].Data.lugar[9] := 3, [26].Data.lugar[10] := 3, [26].Data.lugar[11] := 4, [26].Data.lugar[12] := 4, [26].Data.lugar[13] := 4, [26].Data.lugar[14] := 4, [26].Data.lugar[15] := 3, [26].Data.lugar[16] := 6, [26].Data.flags[0] := 5, [26].Data.flags[1] := 5, [26].Data.flags[2] := 5, [26].Data.flags[3] := 5, [26].Data.flags[4] := 5, [26].Data.flags[5] := 5, [26].Data.flags[6] := 5, [26].Data.flags[7] := 5, [26].Data.flags[8] := 5, [26].Data.flags[9] := 5, [26].Data.flags[10] := 5, [26].Data.flags[11] := 5, [26].Data.flags[12] := 5, [26].Data.flags[13] := 5, [26].Data.flags[14] := 5, [26].Data.flags[15] := 5, [26].Data.flags[16] := 5, [26].Data.fecha_i[0] := 20140324, [26].Data.fecha_i[1] := 20140324, [26].Data.fecha_i[2] := 20140324, [26].Data.fecha_i[3] := 20140324, [26].Data.fecha_i[4] := 20140324, [26].Data.fecha_i[5] := 20140324, [26].Data.fecha_i[6] := 20140324, [26].Data.fecha_i[7] := 20140324, [26].Data.fecha_i[8] := 20140324, [26].Data.fecha_i[9] := 20140324, [26].Data.fecha_i[10] := 20140324, [26].Data.fecha_i[11] := 20140324,
        [26].Data.fecha_i[12] := 20140324, [26].Data.fecha_i[13] := 20140324, [26].Data.fecha_i[14] := 20140324, [26].Data.fecha_i[15] := 20140324, [26].Data.fecha_i[16] := 20140324, [26].Data.fecha_f[0] := 20140324, [26].Data.fecha_f[1] := 20140324, [26].Data.fecha_f[2] := 20140324, [26].Data.fecha_f[3] := 20140324, [26].Data.fecha_f[4] := 20140324, [26].Data.fecha_f[5] := 20140324, [26].Data.fecha_f[6] := 20140324, [26].Data.fecha_f[7] := 20140324, [26].Data.fecha_f[8] := 20140324, [26].Data.fecha_f[9] := 20140324, [26].Data.fecha_f[10] := 20140324, [26].Data.fecha_f[11] := 20140324, [26].Data.fecha_f[12] := 20140324, [26].Data.fecha_f[13] := 20140324, [26].Data.fecha_f[14] := 20140324, [26].Data.fecha_f[15] := 20140324, [26].Data.fecha_f[16] := 20140324, [26].Data.hora_i[0] := 16342414, [26].Data.hora_i[1] := 16344129, [26].Data.hora_i[2] := 16345664, [26].Data.hora_i[3] := 16350589, [26].Data.hora_i[4] := 16342414, [26].Data.hora_i[5] := 16343544, [26].Data.hora_i[6] := 16344669, [26].Data.hora_i[7] := 16345404, [26].Data.hora_i[8] := 16342414, [26].Data.hora_i[9] := 16352739, [26].Data.hora_i[10] := 16362449, [26].Data.hora_i[11] := 16342414, [26].Data.hora_i[12] := 16350629, [26].Data.hora_i[13] := 16360944, [26].Data.hora_i[14] := 16362644, [26].Data.hora_i[15] := 16370269, [26].Data.hora_i[16] := 16373534, [26].Data.hora_f[0] := 16344109, [26].Data.hora_f[1] := 16345644, [26].Data.hora_f[2] := 16350569, [26].Data.hora_f[3] := 16351669, [26].Data.hora_f[4] := 16343524, [26].Data.hora_f[5] := 16344649, [26].Data.hora_f[6] := 16345384, [26].Data.hora_f[7] := 16350119, [26].Data.hora_f[8] := 16352719, [26].Data.hora_f[9] := 16362429, [26].Data.hora_f[10] := 16370249, [26].Data.hora_f[11] := 16350609, [26].Data.hora_f[12] := 16360924, [26].Data.hora_f[13] := 16362624, [26].Data.hora_f[14] := 16363744, [26].Data.hora_f[15] := 16371749, [26].Data.hora_f[16] := 16381729, [27].Head.folio := 39, [27].Head.orden := -3, [27].Head.formula := 'DUMMY$00$00$00$00$00', [27].Head.correlativo := 19,
        [27].Head.total_batch := 20, [27].Head.peso_teorico := 1733.0, [27].Data.codigo[0] := 51, [27].Data.codigo[1] := 53, [27].Data.codigo[2] := 55, [27].Data.codigo[3] := 57, [27].Data.codigo[4] := 60, [27].Data.codigo[5] := 62, [27].Data.codigo[6] := 64, [27].Data.codigo[7] := 66, [27].Data.codigo[8] := 67, [27].Data.codigo[9] := 68, [27].Data.codigo[10] := 69, [27].Data.codigo[11] := 70, [27].Data.codigo[12] := 74, [27].Data.codigo[13] := 75, [27].Data.codigo[14] := 76, [27].Data.codigo[15] := 77, [27].Data.codigo[16] := 81, [27].Data.peso_f[0] := 400.0, [27].Data.peso_f[1] := 350.0, [27].Data.peso_f[2] := 175.0, [27].Data.peso_f[3] := 225.0, [27].Data.peso_f[4] := 125.0, [27].Data.peso_f[5] := 125.0, [27].Data.peso_f[6] := 65.0, [27].Data.peso_f[7] := 65.0, [27].Data.peso_f[8] := 30.0, [27].Data.peso_f[9] := 25.0, [27].Data.peso_f[10] := 17.5, [27].Data.peso_f[11] := 17.5, [27].Data.peso_f[12] := 30.0, [27].Data.peso_f[13] := 5.0, [27].Data.peso_f[14] := 4.0, [27].Data.peso_f[15] := 4.0, [27].Data.peso_f[16] := 70.0, [27].Data.peso_r[0] := 400.74295, [27].Data.peso_r[1] := 350.04123, [27].Data.peso_r[2] := 175.8385, [27].Data.peso_r[3] := 224.96094, [27].Data.peso_r[4] := 124.672356, [27].Data.peso_r[5] := 125.16039, [27].Data.peso_r[6] := 65.37245, [27].Data.peso_r[7] := 65.37756, [27].Data.peso_r[8] := 30.01422, [27].Data.peso_r[9] := 25.012804, [27].Data.peso_r[10] := 17.488533, [27].Data.peso_r[11] := 17.50959, [27].Data.peso_r[12] := 29.994247, [27].Data.peso_r[13] := 4.985035, [27].Data.peso_r[14] := 4.004406, [27].Data.peso_r[15] := 4.0021133, [27].Data.peso_r[16] := 70.10179, [27].Data.tolva[0] := 2, [27].Data.tolva[1] := 4, [27].Data.tolva[2] := 10, [27].Data.tolva[3] := 12, [27].Data.tolva[4] := 7, [27].Data.tolva[5] := 9, [27].Data.tolva[6] := 15,
